RoboDK station: kr30 cnc 071229 table murderer.rdk

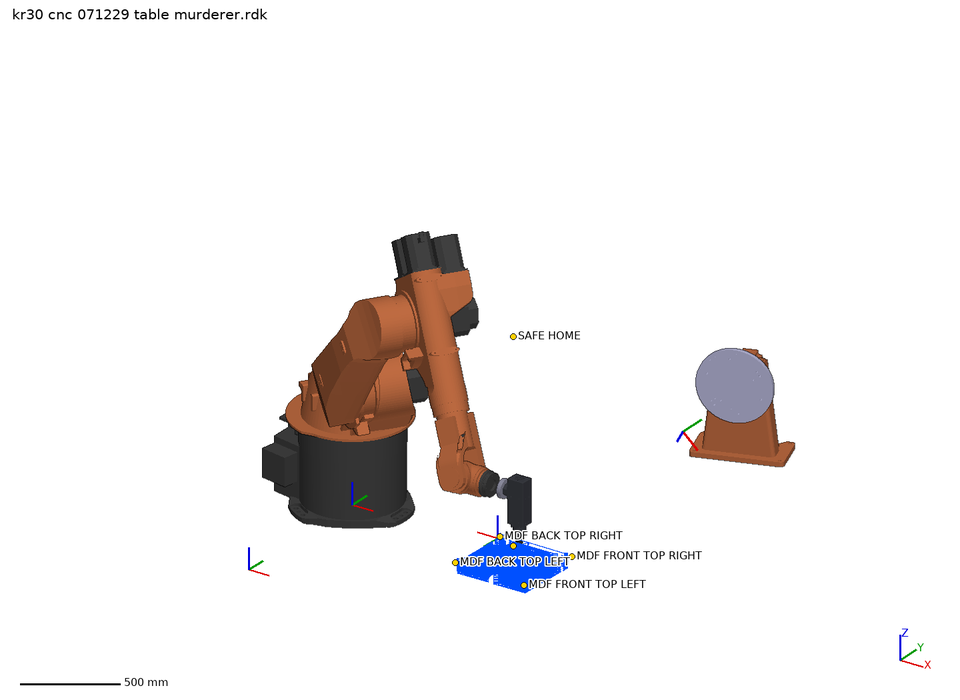
[picture v0: the station drawn from its stored meshes, robots at their saved joint values, targets as dots, program paths as lines]
Station kr30 cnc 071229 table murderer. Poses are relative to the parent item; angles as X-Y-Z fixed-axis rotations.
  - frame GIGASHEEN 7th Axis Base at (0, 1100, 0) mm
    - robot KUKA KP1 MD250: 1 axes, payload 250 kg
        modified DH rows (alpha deg, a mm, theta deg, d mm): 0, 0, 0, 0
        base shift (1750, 1710, 820) mm, rotated rx 0 ry 90 rz -70 deg
        joint limits [-3600] to [3600]; home [0]; saved at [-681.46]
      - frame Reference Rhino at (0, -250, 250) mm
        - object RhinoPart at (0, 0, 0) mm
  - frame GIGASHEEN Base at (0, 2000, 0) mm
    - robot GIGASHEEN (model KUKA KR 30 HA): 6 axes, payload 30 kg, reach 2033 mm, repeatability 0.05 mm, weight 665 kg
        modified DH rows (alpha deg, a mm, theta deg, d mm): 0, 0, 0, 815; -90, 350, 0, 0; 0, 850, -90, 0; -90, 145, 0, 820; 90, 0, 0, 0; -90, 0, 180, 170
        joint limits [-185, -135, -120, -350, -119, -350] to [185, 35, 158, 350, 119, 350]; home [0, -90, 90, 0, 0, 0]; saved at [33.038, -47.483, 104.992, -142.577, 63.826, 162.326]
      - tool 1/2" End Mill TCP, TCP at (337.71, -2.2, 160.57) mm, rotated rx 0 ry 90 rz 0 deg, size 415.8 x 102 x 153.6 mm
    - target MDF BACK TOP LEFT (joint target) at (1355.3, -1043.68, 475.29) mm, rotated rx 179.37 ry 1.37 rz 91.89 deg; joints [27.716, -45.008, 102.25, 116.233, 75.695, -151.59, -681.46] of GIGASHEEN
    - target MDF FRONT TOP LEFT (joint target) at (1780.2, -1054.61, 474.32) mm, rotated rx 179.37 ry 1.37 rz 91.89 deg; joints [22.06, -21.631, 54.581, 104.768, 70.881, -126.376, -681.46] of GIGASHEEN
    - target MDF FRONT TOP RIGHT (joint target) at (1790.65, -653.53, 473.79) mm, rotated rx 179.37 ry 1.37 rz 91.89 deg; joints [10.053, -29.315, 70.245, 98.928, 81.917, -132.341, -681.46] of GIGASHEEN
    - target MDF BACK TOP RIGHT (joint target) at (1365.17, -670.22, 473.91) mm, rotated rx 179.37 ry 1.37 rz 91.89 deg; joints [13.787, -50.344, 113.459, 104.66, 84.215, -154.683, -681.46] of GIGASHEEN
    - target MDF STOCK DEPTH (only use z axis value) (joint target) at (1411.38, -622.96, 416.46) mm, rotated rx 179.37 ry 1.37 rz 91.89 deg; joints [11.502, -45.737, 110.222, 102.707, 85.519, -155.78, -681.46] of GIGASHEEN
    - target SAFE HOME (joint target) at (1411.38, -622.96, 1575.57) mm, rotated rx 179.37 ry 1.37 rz 91.89 deg; joints [11.502, -69.45, 58.776, 88.861, 76.585, -79.989, -681.46] of GIGASHEEN
  - frame Frame 4 at (1373.15, 1298.42, 478.65) mm, rotated rx 1.38 ry 0.62 rz -180 deg
  - machining project Machining Settings: C:/Users/liqui/OneDrive/Documents/GitHub/kuka-fdm/chuck base linearized.apt | rotZ(0) | rotX(0)*rotY(0) | rotz(0)
  - program Machining (9569 instructions, listed below)
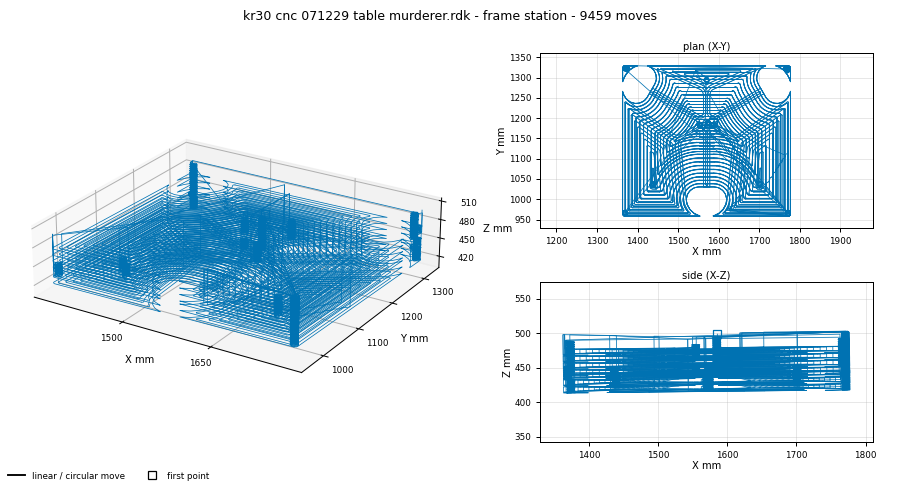
[picture p0: tool path of kr30 cnc 071229 table murderer.rdk in frame station, 9459 of 9459 moves have a stored position in this frame; points joined in program order, loops and branches not executed]

--- program Machining (robot GIGASHEEN) ---
  Accurate (rounding -1 mm)
  Set Ref.: Frame 4
  Set Tool: 1/2" End Mill TCP
  Show 1/2" End Mill TCP
  Print: /'1001'
  Print: /''
  Print: /'Pocket2'
  Set speed (500.0 mm/s)
  Set speed (500.0 mm/s)
  MoveJ 1 to (-212.83, 109.37, 15) mm, rotated rx 180 ry 0 rz 0.01 deg; joints [32.596, -47.797, 105.138, -142.993, 63.549, 162.425]
  MoveL 2 to (-212.83, 109.37, 15) mm, rotated rx 180 ry 0 rz 0.01 deg; joints [32.596, -47.797, 105.138, -142.993, 63.549, 162.425]
  MoveL 3 to (-212.83, 109.37, 15) mm, rotated rx 180 ry 0 rz 0.01 deg; joints [32.596, -47.797, 105.138, -142.993, 63.549, 162.425]
  Set speed (500.0 mm/s)
  MoveL 4 to (-212.83, 109.37, 11.77) mm, rotated rx 180 ry 0 rz 0.01 deg; joints [32.598, -47.633, 105.136, -143.039, 63.679, 162.532]
  Set speed (100.0 mm/s)
  MoveL 5 to (-212.67, 109.35, 11.15) mm, rotated rx -180 ry 0 rz 0.01 deg; joints [32.601, -47.608, 105.149, -143.047, 63.71, 162.556]
  MoveL 6 to (-212.22, 109.32, 10.68) mm, rotated rx -180 ry 0 rz 0.01 deg; joints [32.61, -47.602, 105.184, -143.05, 63.746, 162.58]
  MoveL 7 to (-211.61, 109.34, 10.5) mm, rotated rx 180 ry 0 rz 0.01 deg; joints [32.623, -47.616, 105.231, -143.046, 63.777, 162.596]
  MoveL 8 to (-206.37, 113.36, 10.26) mm, rotated rx -180 ry 0 rz 0.01 deg; joints [32.864, -47.707, 105.436, -142.826, 63.946, 162.558]
  MoveL 9 to (-207.96, 119.77, 10.01) mm, rotated rx -180 ry 0 rz 0.01 deg; joints [33.038, -47.483, 104.992, -142.577, 63.826, 162.326]
  MoveL 10 to (-214.47, 120.88, 9.77) mm, rotated rx -180 ry 0 rz 0.01 deg; joints [32.938, -47.198, 104.43, -142.6, 63.574, 162.187]
  MoveL 11 to (-218.1, 115.37, 9.52) mm, rotated rx -180 ry 0 rz 0.01 deg; joints [32.685, -47.178, 104.424, -142.871, 63.502, 162.318]
  MoveL 12 to (-214.5, 109.83, 9.28) mm, rotated rx 180 ry 0 rz 0.01 deg; joints [32.58, -47.432, 104.981, -143.072, 63.71, 162.572]
  MoveL 13 to (-207.98, 110.91, 9.04) mm, rotated rx 180 ry 0 rz 0.01 deg; joints [32.751, -47.641, 105.433, -142.963, 63.959, 162.653]
  MoveL 14 to (-206.36, 117.31, 8.79) mm, rotated rx 180 ry 0 rz 0.01 deg; joints [32.993, -47.539, 105.238, -142.681, 63.962, 162.476]
  MoveL 15 to (-211.58, 121.36, 8.55) mm, rotated rx 180 ry 0 rz 0.01 deg; joints [33.014, -47.234, 104.629, -142.568, 63.728, 162.261]
  MoveL 16 to (-217.38, 118.21, 8.3) mm, rotated rx -180 ry 0 rz 0.01 deg; joints [32.792, -47.076, 104.336, -142.762, 63.548, 162.276]
  MoveL 17 to (-216.81, 111.63, 8.06) mm, rotated rx 180 ry 0 rz 0.01 deg; joints [32.591, -47.24, 104.709, -143.037, 63.65, 162.513]
  MoveL 18 to (-210.56, 109.51, 7.82) mm, rotated rx 180 ry 0 rz 0.01 deg; joints [32.652, -47.514, 105.301, -143.066, 63.924, 162.697]
  MoveL 19 to (-206.11, 114.39, 7.57) mm, rotated rx -180 ry 0 rz 0.01 deg; joints [32.904, -47.555, 105.402, -142.818, 64.052, 162.618]
  MoveL 20 to (-208.8, 120.42, 7.33) mm, rotated rx 180 ry 0 rz 0.01 deg; joints [33.043, -47.299, 104.891, -142.597, 63.894, 162.38]
  MoveL 21 to (-215.4, 120.37, 7.08) mm, rotated rx 180 ry 0 rz 0.01 deg; joints [32.903, -47.038, 104.379, -142.669, 63.649, 162.277]
  MoveL 22 to (-218.01, 114.3, 6.84) mm, rotated rx 180 ry 0 rz 0.01 deg; joints [32.654, -47.07, 104.481, -142.953, 63.623, 162.444]
  MoveL 23 to (-213.49, 109.49, 6.6) mm, rotated rx -180 ry 0 rz 0.01 deg; joints [32.591, -47.342, 105.073, -143.114, 63.86, 162.689]
  MoveL 24 to (-207.26, 111.7, 6.35) mm, rotated rx 180 ry 0 rz 0.01 deg; joints [32.793, -47.512, 105.446, -142.961, 64.085, 162.728]
  MoveL 25 to (-206.79, 118.29, 6.11) mm, rotated rx 180 ry 0 rz 0.01 deg; joints [33.017, -47.363, 105.152, -142.683, 64.042, 162.526]
  MoveL 26 to (-212.64, 121.36, 5.86) mm, rotated rx -180 ry 0 rz 0.01 deg; joints [32.993, -47.058, 104.543, -142.617, 63.794, 162.332]
  MoveL 27 to (-217.8, 117.23, 5.62) mm, rotated rx 180 ry 0 rz 0.01 deg; joints [32.753, -46.947, 104.349, -142.846, 63.648, 162.39]
  MoveL 28 to (-216.08, 110.85, 5.37) mm, rotated rx -180 ry 0 rz 0.01 deg; joints [32.582, -47.15, 104.802, -143.1, 63.793, 162.64]
  MoveL 29 to (-209.55, 109.87, 5.13) mm, rotated rx -180 ry 0 rz 0.01 deg; joints [32.686, -47.407, 105.358, -143.078, 64.066, 162.791]
  MoveL 30 to (-206.03, 115.46, 4.89) mm, rotated rx 180 ry 0 rz 0.01 deg; joints [32.942, -47.396, 105.351, -142.811, 64.151, 162.673]
  MoveL 31 to (-209.74, 120.92, 4.64) mm, rotated rx 180 ry 0 rz 0.01 deg; joints [33.04, -47.115, 104.789, -142.624, 63.958, 162.437]
  MoveL 32 to (-216.24, 119.71, 4.4) mm, rotated rx -180 ry 0 rz 0.01 deg; joints [32.866, -46.886, 104.344, -142.743, 63.73, 162.374]
  MoveL 33 to (-217.73, 113.27, 4.15) mm, rotated rx -180 ry 0 rz 0.01 deg; joints [32.628, -46.968, 104.55, -143.032, 63.752, 162.571]
  MoveL 34 to (-212.43, 109.33, 3.91) mm, rotated rx 180 ry 0 rz 0.01 deg; joints [32.61, -47.248, 105.159, -143.147, 64.009, 162.8]
  MoveL 35 to (-206.69, 112.6, 3.67) mm, rotated rx 180 ry 0 rz 0.01 deg; joints [32.836, -47.375, 105.441, -142.954, 64.205, 162.797]
  MoveL 36 to (-207.39, 119.17, 3.42) mm, rotated rx 180 ry 0 rz 0.01 deg; joints [33.034, -47.182, 105.057, -142.69, 64.116, 162.576]
  MoveL 37 to (-213.69, 121.16, 3.18) mm, rotated rx 180 ry 0 rz 0.01 deg; joints [32.966, -46.886, 104.468, -142.674, 63.861, 162.41]
  MoveL 38 to (-218.04, 116.19, 2.93) mm, rotated rx 180 ry 0 rz 0.01 deg; joints [32.716, -46.826, 104.378, -142.93, 63.756, 162.509]
  MoveL 39 to (-215.23, 110.21, 2.69) mm, rotated rx -180 ry 0 rz 0.01 deg; joints [32.581, -47.06, 104.896, -143.156, 63.94, 162.764]
  MoveL 40 to (-208.62, 110.4, 2.45) mm, rotated rx -180 ry 0 rz 0.01 deg; joints [32.724, -47.291, 105.399, -143.084, 64.203, 162.877]
  MoveL 41 to (-206.15, 116.52, 2.2) mm, rotated rx -180 ry 0 rz 0.01 deg; joints [32.975, -47.229, 105.285, -142.805, 64.242, 162.725]
  MoveL 42 to (-210.76, 121.24, 1.96) mm, rotated rx -180 ry 0 rz 0.01 deg; joints [33.031, -46.932, 104.689, -142.658, 64.021, 162.498]
  MoveL 43 to (-216.94, 118.9, 1.71) mm, rotated rx -180 ry 0 rz 0.01 deg; joints [32.827, -46.742, 104.326, -142.822, 63.817, 162.477]
  MoveL 44 to (-217.27, 112.31, 1.47) mm, rotated rx 180 ry 0 rz 0.01 deg; joints [32.607, -46.871, 104.63, -143.105, 63.886, 162.699]
  MoveL 45 to (-211.36, 109.36, 1.23) mm, rotated rx -180 ry 0 rz 0.01 deg; joints [32.634, -47.15, 105.236, -143.173, 64.157, 162.905]
  MoveL 46 to (-206.29, 113.59, 0.98) mm, rotated rx 180 ry 0 rz 0.01 deg; joints [32.878, -47.229, 105.418, -142.946, 64.316, 162.86]
  MoveL 47 to (-208.14, 119.93, 0.74) mm, rotated rx 180 ry 0 rz 0.01 deg; joints [33.044, -46.999, 104.957, -142.703, 64.185, 162.626]
  MoveL 48 to (-214.69, 120.78, 0.49) mm, rotated rx -180 ry 0 rz 0.01 deg; joints [32.935, -46.721, 104.404, -142.738, 63.932, 162.494]
  MoveL 49 to (-218.09, 115.12, 0.25) mm, rotated rx -180 ry 0 rz 0.01 deg; joints [32.682, -46.713, 104.423, -143.012, 63.872, 162.632]
  MoveL 50 to (-214.27, 109.74, 0.01) mm, rotated rx 180 ry 0 rz 0.01 deg; joints [32.587, -46.969, 104.989, -143.203, 64.089, 162.883]
  MoveL 51 to (-207.8, 111.08, -0.24) mm, rotated rx 180 ry 0 rz 0.01 deg; joints [32.765, -47.168, 105.424, -143.084, 64.334, 162.957]
  MoveL 52 to (-206.44, 117.54, -0.48) mm, rotated rx 180 ry 0 rz 0.01 deg; joints [33.003, -47.056, 105.206, -142.802, 64.325, 162.775]
  MoveL 53 to (-211.82, 121.38, -0.73) mm, rotated rx 180 ry 0 rz 0.01 deg; joints [33.015, -46.752, 104.595, -142.701, 64.085, 162.563]
  MoveL 54 to (-217.49, 117.99, -0.97) mm, rotated rx -180 ry 0 rz 0.01 deg; joints [32.788, -46.606, 104.324, -142.903, 63.912, 162.586]
  MoveL 55 to (-216.66, 111.44, -1.21) mm, rotated rx -180 ry 0 rz 0.01 deg; joints [32.593, -46.778, 104.716, -143.173, 64.026, 162.826]
  MoveL 56 to (-210.32, 109.58, -1.46) mm, rotated rx -180 ry 0 rz 0.01 deg; joints [32.665, -47.046, 105.302, -143.19, 64.302, 163.004]
  MoveL 57 to (-206.07, 114.63, -1.7) mm, rotated rx 180 ry 0 rz 0.01 deg; joints [32.918, -47.075, 105.378, -142.937, 64.42, 162.917]
  MoveL 58 to (-209.01, 120.55, -1.95) mm, rotated rx 180 ry 0 rz 0.01 deg; joints [33.048, -46.815, 104.853, -142.723, 64.251, 162.679]
  MoveL 59 to (-215.6, 120.23, -2.19) mm, rotated rx -180 ry 0 rz 0.01 deg; joints [32.9, -46.562, 104.356, -142.807, 64.008, 162.584]
  MoveL 60 to (-217.96, 114.06, -2.43) mm, rotated rx 180 ry 0 rz 0.01 deg; joints [32.652, -46.605, 104.481, -143.093, 63.995, 162.757]
  MoveL 61 to (-213.25, 109.44, -2.68) mm, rotated rx -180 ry 0 rz 0.01 deg; joints [32.6, -46.877, 105.079, -143.242, 64.239, 162.998]
  MoveL 62 to (-207.12, 111.9, -2.92) mm, rotated rx -180 ry 0 rz 0.01 deg; joints [32.808, -47.036, 105.431, -143.079, 64.459, 163.03]
  MoveL 63 to (-206.92, 118.5, -3.17) mm, rotated rx -180 ry 0 rz 0.01 deg; joints [33.026, -46.878, 105.116, -142.804, 64.403, 162.823]
  MoveL 64 to (-212.89, 121.33, -3.41) mm, rotated rx 180 ry 0 rz 0.01 deg; joints [32.992, -46.576, 104.51, -142.751, 64.149, 162.635]
  MoveL 65 to (-217.87, 116.99, -3.65) mm, rotated rx -180 ry 0 rz 0.01 deg; joints [32.749, -46.478, 104.339, -142.986, 64.013, 162.701]
  MoveL 66 to (-215.9, 110.69, -3.9) mm, rotated rx -180 ry 0 rz 0.01 deg; joints [32.586, -46.686, 104.808, -143.233, 64.17, 162.951]
  MoveL 67 to (-209.33, 109.97, -4.14) mm, rotated rx -180 ry 0 rz 0.01 deg; joints [32.7, -46.935, 105.353, -143.199, 64.443, 163.095]
  MoveL 68 to (-206.04, 115.7, -4.39) mm, rotated rx -180 ry 0 rz 0.01 deg; joints [32.954, -46.913, 105.321, -142.929, 64.516, 162.971]
  MoveL 69 to (-209.97, 121.01, -4.63) mm, rotated rx 180 ry 0 rz 0.01 deg; joints [33.044, -46.63, 104.75, -142.751, 64.314, 162.736]
  MoveL 70 to (-216.41, 119.53, -4.87) mm, rotated rx -180 ry 0 rz 0.01 deg; joints [32.862, -46.411, 104.322, -142.882, 64.09, 162.681]
  MoveL 71 to (-217.64, 113.05, -5.12) mm, rotated rx -180 ry 0 rz 0.01 deg; joints [32.627, -46.503, 104.551, -143.169, 64.124, 162.883]
  MoveL 72 to (-212.19, 109.32, -5.36) mm, rotated rx -180 ry 0 rz 0.01 deg; joints [32.62, -46.781, 105.161, -143.273, 64.388, 163.107]
  MoveL 73 to (-206.59, 112.82, -5.61) mm, rotated rx 180 ry 0 rz 0.01 deg; joints [32.85, -46.896, 105.42, -143.071, 64.576, 163.096]
  MoveL 74 to (-207.55, 119.35, -5.85) mm, rotated rx -180 ry 0 rz 0.01 deg; joints [33.042, -46.696, 105.018, -142.812, 64.474, 162.872]
  MoveL 75 to (-213.92, 121.09, -6.1) mm, rotated rx -180 ry 0 rz 0.01 deg; joints [32.964, -46.405, 104.435, -142.808, 64.217, 162.712]
  MoveL 76 to (-218.07, 115.95, -6.34) mm, rotated rx -180 ry 0 rz 0.01 deg; joints [32.713, -46.358, 104.37, -143.068, 64.123, 162.819]
  MoveL 77 to (-215.02, 110.09, -6.58) mm, rotated rx 180 ry 0 rz 0.01 deg; joints [32.587, -46.595, 104.9, -143.286, 64.317, 163.073]
  MoveL 78 to (-208.43, 110.54, -6.83) mm, rotated rx -180 ry 0 rz 0.01 deg; joints [32.738, -46.817, 105.389, -143.202, 64.578, 163.179]
  MoveL 79 to (-206.2, 116.76, -7.07) mm, rotated rx 180 ry 0 rz 0.01 deg; joints [32.987, -46.744, 105.25, -142.923, 64.604, 163.021]
  MoveL 80 to (-211, 121.29, -7.32) mm, rotated rx 180 ry 0 rz 0.01 deg; joints [33.033, -46.447, 104.649, -142.787, 64.376, 162.796]
  MoveL 81 to (-217.08, 118.7, -7.56) mm, rotated rx -180 ry 0 rz 0.01 deg; joints [32.823, -46.268, 104.306, -142.96, 64.178, 162.784]
  MoveL 82 to (-217.15, 112.1, -7.8) mm, rotated rx -180 ry 0 rz 0.01 deg; joints [32.608, -46.406, 104.631, -143.24, 64.26, 163.009]
  MoveL 83 to (-211.12, 109.39, -8.05) mm, rotated rx -180 ry 0 rz 0.01 deg; joints [32.646, -46.68, 105.234, -143.295, 64.535, 163.21]
  MoveL 84 to (-206.23, 113.83, -8.29) mm, rotated rx -180 ry 0 rz 0.01 deg; joints [32.892, -46.748, 105.392, -143.062, 64.684, 163.157]
  MoveL 85 to (-208.33, 120.09, -8.54) mm, rotated rx -180 ry 0 rz 0.01 deg; joints [33.051, -46.512, 104.914, -142.826, 64.541, 162.922]
  MoveL 86 to (-214.91, 120.67, -8.78) mm, rotated rx -180 ry 0 rz 0.01 deg; joints [32.932, -46.241, 104.373, -142.872, 64.288, 162.796]
  MoveL 87 to (-218.08, 114.88, -9.02) mm, rotated rx -180 ry 0 rz 0.01 deg; joints [32.679, -46.244, 104.416, -143.15, 64.24, 162.941]
  MoveL 88 to (-214.04, 109.65, -9.27) mm, rotated rx 180 ry 0 rz 0.01 deg; joints [32.594, -46.503, 104.991, -143.331, 64.466, 163.191]
  MoveL 89 to (-207.64, 111.25, -9.51) mm, rotated rx 180 ry 0 rz 0.01 deg; joints [32.78, -46.691, 105.408, -143.2, 64.707, 163.256]
  MoveL 90 to (-206.54, 117.77, -9.76) mm, rotated rx -180 ry 0 rz 0.01 deg; joints [33.014, -46.569, 105.167, -142.92, 64.685, 163.069]
  MoveL 91 to (-212.06, 121.38, -10) mm, rotated rx -180 ry 0 rz 0.01 deg; joints [33.015, -46.268, 104.555, -142.83, 64.439, 162.862]
  MoveL 92 to (-213.99, 121.38, -10) mm, rotated rx -180 ry 0 rz 0.01 deg; joints [32.975, -46.196, 104.405, -142.85, 64.364, 162.828]
  MoveC 93 to (-215.91, 120.27, -10) mm, rotated rx 180 ry 0 rz 0.01 deg; joints [32.899, -46.15, 104.311, -142.916, 64.301, 162.831] to (-215.92, 118.06, -10) mm, rotated rx -180 ry 0 rz 0.01 deg; joints [32.827, -46.201, 104.423, -143.008, 64.326, 162.905]
  MoveL 94 to (-214.81, 116.14, -10) mm, rotated rx -180 ry 0 rz 0.01 deg; joints [32.788, -46.287, 104.605, -143.077, 64.391, 162.988]
  MoveC 95 to (-213.77, 115.1, -10) mm, rotated rx 180 ry 0 rz 0.01 deg; joints [32.776, -46.35, 104.738, -143.11, 64.444, 163.04] to (-212.35, 114.72, -10) mm, rotated rx 180 ry 0 rz 0.01 deg; joints [32.794, -46.412, 104.868, -143.111, 64.504, 163.077]
  MoveL 96 to (-181.15, 114.72, -10) mm, rotated rx 180 ry 0 rz 0.01 deg; joints [33.456, -47.555, 107.262, -142.767, 65.707, 163.609]
  MoveC 97 to (-179.73, 115.1, -10) mm, rotated rx 180 ry 0 rz 0.01 deg; joints [33.499, -47.597, 107.35, -142.735, 65.756, 163.62] to (-178.69, 116.13, -10) mm, rotated rx -180 ry 0 rz 0.01 deg; joints [33.555, -47.611, 107.377, -142.679, 65.784, 163.604]
  MoveL 98 to (-177.58, 118.05, -10) mm, rotated rx 180 ry 0 rz 0.01 deg; joints [33.642, -47.607, 107.365, -142.587, 65.804, 163.561]
  MoveC 99 to (-177.58, 120.27, -10) mm, rotated rx -180 ry 0 rz 0.01 deg; joints [33.714, -47.556, 107.253, -142.495, 65.778, 163.489] to (-179.5, 121.38, -10) mm, rotated rx -180 ry 0 rz 0.01 deg; joints [33.709, -47.461, 107.052, -142.471, 65.692, 163.42]
  MoveL 100 to (-212.06, 121.38, -10) mm, rotated rx -180 ry 0 rz 0.01 deg; joints [33.015, -46.268, 104.555, -142.83, 64.439, 162.862]
  MoveC 101 to (-215.55, 122.47, -10) mm, rotated rx 180 ry 0 rz 0.01 deg; joints [32.977, -46.112, 104.229, -142.82, 64.29, 162.765] to (-217.79, 125.34, -10) mm, rotated rx -180 ry 0 rz 0.01 deg; joints [33.023, -45.961, 103.908, -142.723, 64.17, 162.63]
  MoveC 102 to (-219.97, 128.24, -10) mm, rotated rx 180 ry 0 rz 0.01 deg; joints [33.07, -45.812, 103.59, -142.624, 64.051, 162.494] to (-223.36, 129.52, -10) mm, rotated rx 180 ry 0 rz 0.01 deg; joints [33.04, -45.654, 103.259, -142.603, 63.904, 162.391]
  MoveC 103 to (-226.44, 129.78, -10) mm, rotated rx -180 ry 0 rz 0.01 deg; joints [32.985, -45.532, 103.004, -142.622, 63.78, 162.327] to (-229.51, 130.08, -10) mm, rotated rx -180 ry 0 rz 0.01 deg; joints [32.931, -45.409, 102.747, -142.639, 63.656, 162.262]
  MoveC 104 to (-231.31, 129.16, -10) mm, rotated rx -180 ry 0 rz 0.01 deg; joints [32.865, -45.362, 102.651, -142.694, 63.595, 162.26] to (-231.22, 127.14, -10) mm, rotated rx 180 ry 0 rz 0.01 deg; joints [32.802, -45.413, 102.762, -142.778, 63.622, 162.331]
  MoveC 105 to (-228.51, 123.21, -10) mm, rotated rx 180 ry 0 rz 0.01 deg; joints [32.733, -45.608, 103.175, -142.916, 63.773, 162.511] to (-225.92, 119.21, -10) mm, rotated rx 180 ry 0 rz 0.01 deg; joints [32.657, -45.799, 103.581, -143.059, 63.921, 162.691]
  MoveC 106 to (-223.44, 115.14, -10) mm, rotated rx 180 ry 0 rz 0.01 deg; joints [32.578, -45.987, 103.981, -143.205, 64.065, 162.87] to (-221.02, 111.03, -10) mm, rotated rx -180 ry 0 rz 0.01 deg; joints [32.495, -46.173, 104.375, -143.353, 64.206, 163.048]
  MoveC 107 to (-217.92, 107.92, -10) mm, rotated rx 180 ry 0 rz 0.01 deg; joints [32.458, -46.36, 104.773, -143.452, 64.363, 163.204] to (-213.68, 106.78, -10) mm, rotated rx 180 ry 0 rz 0.01 deg; joints [32.509, -46.544, 105.16, -143.457, 64.542, 163.315]
  MoveL 108 to (-179.84, 106.78, -10) mm, rotated rx 180 ry 0 rz 0.01 deg; joints [33.224, -47.784, 107.756, -143.082, 65.848, 163.886]
  MoveC 109 to (-175.59, 107.92, -10) mm, rotated rx 180 ry 0 rz 0.01 deg; joints [33.353, -47.911, 108.021, -142.983, 65.997, 163.92] to (-172.48, 111.03, -10) mm, rotated rx -180 ry 0 rz 0.01 deg; joints [33.523, -47.951, 108.1, -142.817, 66.079, 163.872]
  MoveC 110 to (-170.06, 115.13, -10) mm, rotated rx 180 ry 0 rz 0.01 deg; joints [33.71, -47.944, 108.076, -142.617, 66.123, 163.78] to (-167.6, 119.21, -10) mm, rotated rx 180 ry 0 rz 0.01 deg; joints [33.898, -47.938, 108.057, -142.418, 66.168, 163.69]
  MoveC 111 to (-165.03, 123.22, -10) mm, rotated rx 180 ry 0 rz 0.01 deg; joints [34.086, -47.937, 108.047, -142.22, 66.219, 163.603] to (-162.31, 127.14, -10) mm, rotated rx 180 ry 0 rz 0.01 deg; joints [34.273, -47.942, 108.051, -142.024, 66.275, 163.522]
  MoveC 112 to (-162.21, 129.16, -10) mm, rotated rx 180 ry 0 rz 0.01 deg; joints [34.342, -47.899, 107.956, -141.94, 66.256, 163.458] to (-164.01, 130.09, -10) mm, rotated rx -180 ry 0 rz 0.01 deg; joints [34.332, -47.813, 107.775, -141.924, 66.177, 163.398]
  MoveC 113 to (-167.84, 129.69, -10) mm, rotated rx -180 ry 0 rz 0.01 deg; joints [34.234, -47.685, 107.508, -141.987, 66.038, 163.346] to (-171.67, 129.27, -10) mm, rotated rx 180 ry 0 rz 0.01 deg; joints [34.136, -47.558, 107.243, -142.051, 65.898, 163.295]
  MoveC 114 to (-175.51, 128.94, -10) mm, rotated rx -180 ry 0 rz 0.01 deg; joints [34.041, -47.428, 106.97, -142.111, 65.756, 163.241] to (-179.36, 128.83, -10) mm, rotated rx 180 ry 0 rz 0.01 deg; joints [33.954, -47.292, 106.685, -142.161, 65.611, 163.179]
  MoveL 115 to (-205.63, 128.84, -10) mm, rotated rx -180 ry 0 rz 0.01 deg; joints [33.39, -46.332, 104.676, -142.453, 64.603, 162.727]
  MoveC 116 to (-214.5, 129.01, -10) mm, rotated rx -180 ry 0 rz 0.01 deg; joints [33.209, -45.998, 103.978, -142.537, 64.256, 162.565] to (-223.36, 129.52, -10) mm, rotated rx -180 ry 0 rz 0.01 deg; joints [33.04, -45.654, 103.259, -142.603, 63.904, 162.391]
  MoveC 117 to (-226.59, 130.78, -10) mm, rotated rx 180 ry 0 rz 0.01 deg; joints [33.014, -45.502, 102.941, -142.582, 63.763, 162.29] to (-228.56, 133.63, -10) mm, rotated rx -180 ry 0 rz 0.01 deg; joints [33.063, -45.36, 102.639, -142.482, 63.652, 162.159]
  MoveC 118 to (-230.49, 136.49, -10) mm, rotated rx -180 ry 0 rz 0.01 deg; joints [33.114, -45.219, 102.34, -142.38, 63.544, 162.026] to (-233.65, 137.88, -10) mm, rotated rx -180 ry 0 rz 0.01 deg; joints [33.093, -45.066, 102.018, -142.351, 63.403, 161.922]
  MoveC 119 to (-239.01, 138.68, -10) mm, rotated rx -180 ry 0 rz 0.01 deg; joints [33.008, -44.842, 101.55, -142.365, 63.182, 161.796] to (-244.35, 139.65, -10) mm, rotated rx 180 ry 0 rz 0.01 deg; joints [32.93, -44.614, 101.074, -142.371, 62.958, 161.664]
  MoveC 120 to (-245.19, 139.83, -10) mm, rotated rx 180 ry 0 rz 0.01 deg; joints [32.918, -44.577, 100.997, -142.371, 62.923, 161.642] to (-246.02, 140.03, -10) mm, rotated rx 180 ry 0 rz 0.01 deg; joints [32.908, -44.54, 100.92, -142.37, 62.888, 161.62]
  MoveC 121 to (-246.85, 140.23, -10) mm, rotated rx -180 ry 0 rz 0.01 deg; joints [32.897, -44.504, 100.843, -142.368, 62.852, 161.597] to (-247.69, 140.41, -10) mm, rotated rx 180 ry 0 rz 0.01 deg; joints [32.886, -44.467, 100.766, -142.368, 62.817, 161.576]
  MoveC 122 to (-249.42, 139.63, -10) mm, rotated rx -180 ry 0 rz 0.01 deg; joints [32.826, -44.419, 100.667, -142.415, 62.756, 161.57] to (-249.25, 137.73, -10) mm, rotated rx -180 ry 0 rz 0.01 deg; joints [32.77, -44.471, 100.779, -142.493, 62.784, 161.639]
  MoveC 123 to (-245.42, 133.29, -10) mm, rotated rx 180 ry 0 rz 0.01 deg; joints [32.708, -44.725, 101.316, -142.647, 62.988, 161.863] to (-241.53, 128.89, -10) mm, rotated rx 180 ry 0 rz 0.01 deg; joints [32.647, -44.979, 101.852, -142.798, 63.193, 162.084]
  MoveC 124 to (-237.77, 124.39, -10) mm, rotated rx -180 ry 0 rz 0.01 deg; joints [32.58, -45.229, 102.382, -142.953, 63.394, 162.306] to (-234.3, 119.65, -10) mm, rotated rx 180 ry 0 rz 0.01 deg; joints [32.5, -45.472, 102.897, -143.12, 63.585, 162.527]
  MoveC 125 to (-231.84, 115.78, -10) mm, rotated rx -180 ry 0 rz 0.01 deg; joints [32.426, -45.656, 103.287, -143.259, 63.726, 162.701] to (-229.63, 111.75, -10) mm, rotated rx 180 ry 0 rz 0.01 deg; joints [32.341, -45.832, 103.663, -143.407, 63.859, 162.874]
  MoveC 126 to (-227.51, 107.68, -10) mm, rotated rx -180 ry 0 rz 0.01 deg; joints [32.254, -46.006, 104.033, -143.557, 63.989, 163.046] to (-225.27, 103.68, -10) mm, rotated rx 180 ry 0 rz 0.01 deg; joints [32.169, -46.181, 104.407, -143.703, 64.123, 163.216]
  MoveC 127 to (-222.17, 100.57, -10) mm, rotated rx 180 ry 0 rz 0.01 deg; joints [32.132, -46.369, 104.804, -143.803, 64.28, 163.372] to (-217.92, 99.43, -10) mm, rotated rx 180 ry 0 rz 0.01 deg; joints [32.182, -46.553, 105.192, -143.808, 64.46, 163.482]
  MoveL 128 to (-175.6, 99.43, -10) mm, rotated rx -180 ry 0 rz 0.01 deg; joints [33.073, -48.102, 108.438, -143.337, 66.094, 164.191]
  MoveC 129 to (-171.35, 100.57, -10) mm, rotated rx 180 ry 0 rz 0.01 deg; joints [33.202, -48.229, 108.702, -143.237, 66.243, 164.224] to (-168.24, 103.68, -10) mm, rotated rx -180 ry 0 rz 0.01 deg; joints [33.373, -48.27, 108.783, -143.07, 66.324, 164.176]
  MoveC 130 to (-164.24, 110.52, -10) mm, rotated rx -180 ry 0 rz 0.01 deg; joints [33.687, -48.257, 108.743, -142.736, 66.396, 164.024] to (-160.18, 117.33, -10) mm, rotated rx 180 ry 0 rz 0.01 deg; joints [34, -48.245, 108.705, -142.403, 66.47, 163.873]
  MoveC 131 to (-155.83, 123.97, -10) mm, rotated rx 180 ry 0 rz 0.01 deg; joints [34.314, -48.245, 108.694, -142.073, 66.555, 163.732] to (-150.99, 130.25, -10) mm, rotated rx -180 ry 0 rz 0.01 deg; joints [34.628, -48.269, 108.733, -141.751, 66.662, 163.609]
  MoveC 132 to (-149.35, 132.16, -10) mm, rotated rx 180 ry 0 rz 0.01 deg; joints [34.727, -48.282, 108.757, -141.652, 66.701, 163.575] to (-147.65, 134.01, -10) mm, rotated rx -180 ry 0 rz 0.01 deg; joints [34.826, -48.299, 108.787, -141.553, 66.743, 163.543]
  MoveC 133 to (-145.94, 135.85, -10) mm, rotated rx 180 ry 0 rz 0.01 deg; joints [34.924, -48.315, 108.819, -141.455, 66.785, 163.512] to (-144.26, 137.72, -10) mm, rotated rx -180 ry 0 rz 0.01 deg; joints [35.023, -48.33, 108.847, -141.356, 66.825, 163.479]
  MoveC 134 to (-144.06, 139.61, -10) mm, rotated rx 180 ry 0 rz 0.01 deg; joints [35.089, -48.292, 108.764, -141.276, 66.81, 163.421] to (-145.78, 140.42, -10) mm, rotated rx 180 ry 0 rz 0.01 deg; joints [35.076, -48.213, 108.596, -141.266, 66.737, 163.366]
  MoveC 135 to (-154.12, 138.92, -10) mm, rotated rx 180 ry 0 rz 0.01 deg; joints [34.839, -47.955, 108.058, -141.435, 66.444, 163.276] to (-162.48, 137.5, -10) mm, rotated rx -180 ry 0 rz 0.01 deg; joints [34.606, -47.693, 107.51, -141.599, 66.149, 163.181]
  MoveC 136 to (-170.89, 136.46, -10) mm, rotated rx -180 ry 0 rz 0.01 deg; joints [34.386, -47.417, 106.933, -141.745, 65.844, 163.073] to (-179.36, 136.12, -10) mm, rotated rx -180 ry 0 rz 0.01 deg; joints [34.189, -47.12, 106.313, -141.86, 65.527, 162.94]
  MoveL 137 to (-211.94, 136.31, -10) mm, rotated rx -180 ry 0 rz 0.01 deg; joints [33.495, -45.921, 103.804, -142.207, 64.272, 162.365]
  MoveC 138 to (-222.82, 136.77, -10) mm, rotated rx -180 ry 0 rz 0.01 deg; joints [33.282, -45.502, 102.93, -142.296, 63.842, 162.156] to (-233.65, 137.88, -10) mm, rotated rx -180 ry 0 rz 0.01 deg; joints [33.093, -45.066, 102.018, -142.351, 63.403, 161.922]
  MoveC 139 to (-236.39, 139.14, -10) mm, rotated rx -180 ry 0 rz 0.01 deg; joints [33.076, -44.931, 101.735, -142.323, 63.281, 161.828] to (-237.97, 141.71, -10) mm, rotated rx 180 ry 0 rz 0.01 deg; joints [33.125, -44.809, 101.477, -142.23, 63.189, 161.711]
  MoveC 140 to (-239.5, 144.29, -10) mm, rotated rx -180 ry 0 rz 0.01 deg; joints [33.175, -44.688, 101.22, -142.135, 63.099, 161.594] to (-242.17, 145.66, -10) mm, rotated rx 180 ry 0 rz 0.01 deg; joints [33.163, -44.553, 100.935, -142.101, 62.977, 161.497]
  MoveC 141 to (-243.73, 145.98, -10) mm, rotated rx -180 ry 0 rz 0.01 deg; joints [33.141, -44.485, 100.794, -142.101, 62.911, 161.457] to (-245.29, 146.31, -10) mm, rotated rx 180 ry 0 rz 0.01 deg; joints [33.119, -44.417, 100.651, -142.1, 62.845, 161.416]
  MoveC 142 to (-260.07, 150.25, -10) mm, rotated rx -180 ry 0 rz 0.01 deg; joints [32.943, -43.747, 99.251, -142.054, 62.208, 160.998] to (-274.43, 155.48, -10) mm, rotated rx 180 ry 0 rz 0.01 deg; joints [32.817, -43.05, 97.796, -141.937, 61.566, 160.532]
  MoveC 143 to (-275.99, 154.95, -10) mm, rotated rx 180 ry 0 rz 0.01 deg; joints [32.77, -43.002, 97.695, -141.97, 61.508, 160.521] to (-275.66, 153.34, -10) mm, rotated rx -180 ry 0 rz 0.01 deg; joints [32.727, -43.055, 97.808, -142.036, 61.54, 160.585]
  MoveC 144 to (-256.3, 136, -10) mm, rotated rx -180 ry 0 rz 0.01 deg; joints [32.573, -44.239, 100.3, -142.623, 62.521, 161.567] to (-239.99, 115.76, -10) mm, rotated rx -180 ry 0 rz 0.01 deg; joints [32.26, -45.346, 102.641, -143.335, 63.403, 162.556]
  MoveC 145 to (-237.06, 111.16, -10) mm, rotated rx -180 ry 0 rz 0.01 deg; joints [32.171, -45.564, 103.104, -143.501, 63.572, 162.762] to (-234.44, 106.38, -10) mm, rotated rx -180 ry 0 rz 0.01 deg; joints [32.07, -45.773, 103.55, -143.678, 63.73, 162.967]
  MoveC 146 to (-231.91, 101.55, -10) mm, rotated rx 180 ry 0 rz 0.01 deg; joints [31.965, -45.979, 103.989, -143.857, 63.885, 163.171] to (-229.25, 96.79, -10) mm, rotated rx -180 ry 0 rz 0.01 deg; joints [31.864, -46.188, 104.432, -144.031, 64.044, 163.373]
  MoveC 147 to (-226.15, 93.68, -10) mm, rotated rx -180 ry 0 rz 0.01 deg; joints [31.826, -46.374, 104.829, -144.131, 64.201, 163.528] to (-221.9, 92.54, -10) mm, rotated rx 180 ry 0 rz 0.01 deg; joints [31.875, -46.559, 105.217, -144.137, 64.382, 163.637]
  MoveL 148 to (-171.62, 92.54, -10) mm, rotated rx 180 ry 0 rz 0.01 deg; joints [32.93, -48.399, 109.074, -143.575, 66.325, 164.473]
  MoveC 149 to (-167.37, 93.68, -10) mm, rotated rx 180 ry 0 rz 0.01 deg; joints [33.06, -48.525, 109.337, -143.475, 66.473, 164.506] to (-164.26, 96.79, -10) mm, rotated rx -180 ry 0 rz 0.01 deg; joints [33.231, -48.566, 109.418, -143.306, 66.554, 164.459]
  MoveL 150 to (-155.69, 111.78, -10) mm, rotated rx -180 ry 0 rz 0.01 deg; joints [33.917, -48.531, 109.316, -142.575, 66.703, 164.124]
  MoveC 151 to (-151.1, 119.11, -10) mm, rotated rx 180 ry 0 rz 0.01 deg; joints [34.261, -48.524, 109.289, -142.212, 66.789, 163.966] to (-145.88, 125.99, -10) mm, rotated rx -180 ry 0 rz 0.01 deg; joints [34.604, -48.548, 109.327, -141.86, 66.903, 163.831]
  MoveC 152 to (-139.41, 133.39, -10) mm, rotated rx -180 ry 0 rz 0.01 deg; joints [34.993, -48.601, 109.424, -141.469, 67.055, 163.7] to (-132.6, 140.47, -10) mm, rotated rx -180 ry 0 rz 0.01 deg; joints [35.38, -48.671, 109.557, -141.086, 67.223, 163.583]
  MoveC 153 to (-125.4, 147.16, -10) mm, rotated rx -180 ry 0 rz 0.01 deg; joints [35.764, -48.76, 109.733, -140.712, 67.407, 163.485] to (-117.79, 153.38, -10) mm, rotated rx 180 ry 0 rz 0.01 deg; joints [36.144, -48.872, 109.956, -140.35, 67.611, 163.408]
  MoveC 154 to (-117.47, 154.99, -10) mm, rotated rx -180 ry 0 rz 0.01 deg; joints [36.203, -48.844, 109.894, -140.28, 67.603, 163.361] to (-119.03, 155.51, -10) mm, rotated rx 180 ry 0 rz 0.01 deg; joints [36.183, -48.778, 109.755, -140.281, 67.54, 163.318]
  MoveC 155 to (-144.72, 147.15, -10) mm, rotated rx 180 ry 0 rz 0.01 deg; joints [35.318, -48.09, 108.325, -140.975, 66.697, 163.164] to (-171.45, 143.25, -10) mm, rotated rx -180 ry 0 rz 0.01 deg; joints [34.592, -47.236, 106.542, -141.472, 65.744, 162.839]
  MoveL 156 to (-214.92, 143.01, -10) mm, rotated rx -180 ry 0 rz 0.01 deg; joints [33.646, -45.649, 103.226, -141.959, 64.08, 162.086]
  MoveC 157 to (-228.61, 143.68, -10) mm, rotated rx 180 ry 0 rz 0.01 deg; joints [33.38, -45.118, 102.117, -142.063, 63.536, 161.815] to (-242.17, 145.66, -10) mm, rotated rx 180 ry 0 rz 0.01 deg; joints [33.163, -44.553, 100.935, -142.101, 62.977, 161.497]
  MoveC 158 to (-244.83, 147.08, -10) mm, rotated rx 180 ry 0 rz 0.01 deg; joints [33.153, -44.416, 100.648, -142.064, 62.854, 161.398] to (-246.26, 149.74, -10) mm, rotated rx -180 ry 0 rz 0.01 deg; joints [33.207, -44.296, 100.394, -141.965, 62.767, 161.278]
  MoveC 159 to (-247.64, 152.41, -10) mm, rotated rx 180 ry 0 rz 0.01 deg; joints [33.262, -44.177, 100.142, -141.865, 62.682, 161.159] to (-250.24, 153.93, -10) mm, rotated rx 180 ry 0 rz 0.01 deg; joints [33.256, -44.039, 99.853, -141.822, 62.561, 161.056]
  MoveC 160 to (-267.07, 159.34, -10) mm, rotated rx -180 ry 0 rz 0.01 deg; joints [33.083, -43.247, 98.196, -141.723, 61.821, 160.539] to (-283.1, 166.79, -10) mm, rotated rx 180 ry 0 rz 0.01 deg; joints [32.992, -42.42, 96.47, -141.516, 61.082, 159.95]
  MoveC 161 to (-285.35, 166.74, -10) mm, rotated rx 180 ry 0 rz 0.01 deg; joints [32.946, -42.331, 96.285, -141.532, 60.991, 159.906] to (-286.46, 164.79, -10) mm, rotated rx 180 ry 0 rz 0.01 deg; joints [32.865, -42.336, 96.298, -141.621, 60.967, 159.955]
  MoveL 162 to (-286.46, 156.66, -10) mm, rotated rx 180 ry 0 rz 0.01 deg; joints [32.616, -42.54, 96.735, -141.966, 61.06, 160.251]
  MoveC 163 to (-285.7, 153.53, -10) mm, rotated rx 180 ry 0 rz 0.01 deg; joints [32.535, -42.648, 96.965, -142.094, 61.127, 160.379] to (-283.59, 151.1, -10) mm, rotated rx 180 ry 0 rz 0.01 deg; joints [32.502, -42.793, 97.269, -142.183, 61.241, 160.508]
  MoveC 164 to (-262.73, 133.3, -10) mm, rotated rx 180 ry 0 rz 0.01 deg; joints [32.36, -44.053, 99.917, -142.787, 62.293, 161.54] to (-245.34, 112.1, -10) mm, rotated rx -180 ry 0 rz 0.01 deg; joints [32.035, -45.226, 102.397, -143.536, 63.231, 162.583]
  MoveC 165 to (-241.98, 106.82, -10) mm, rotated rx 180 ry 0 rz 0.01 deg; joints [31.933, -45.476, 102.929, -143.728, 63.425, 162.82] to (-238.96, 101.32, -10) mm, rotated rx -180 ry 0 rz 0.01 deg; joints [31.816, -45.717, 103.441, -143.932, 63.607, 163.055]
  MoveC 166 to (-236.05, 95.78, -10) mm, rotated rx -180 ry 0 rz 0.01 deg; joints [31.694, -45.953, 103.944, -144.138, 63.786, 163.289] to (-233, 90.31, -10) mm, rotated rx 180 ry 0 rz 0.01 deg; joints [31.577, -46.192, 104.453, -144.34, 63.968, 163.52]
  MoveC 167 to (-229.89, 87.2, -10) mm, rotated rx 180 ry 0 rz 0.01 deg; joints [31.538, -46.378, 104.848, -144.44, 64.127, 163.674] to (-225.65, 86.06, -10) mm, rotated rx -180 ry 0 rz 0.01 deg; joints [31.586, -46.563, 105.237, -144.447, 64.307, 163.783]
  MoveL 168 to (-167.88, 86.06, -10) mm, rotated rx -180 ry 0 rz 0.01 deg; joints [32.794, -48.676, 109.668, -143.799, 66.542, 164.737]
  MoveC 169 to (-163.63, 87.2, -10) mm, rotated rx 180 ry 0 rz 0.01 deg; joints [32.924, -48.802, 109.931, -143.698, 66.689, 164.769] to (-160.52, 90.31, -10) mm, rotated rx -180 ry 0 rz 0.01 deg; joints [33.096, -48.843, 110.013, -143.529, 66.771, 164.722]
  MoveC 170 to (-155.91, 98.38, -10) mm, rotated rx -180 ry 0 rz 0.01 deg; joints [33.467, -48.826, 109.962, -143.134, 66.85, 164.544] to (-151.38, 106.49, -10) mm, rotated rx -180 ry 0 rz 0.01 deg; joints [33.838, -48.803, 109.898, -142.738, 66.926, 164.362]
  MoveC 171 to (-146.5, 114.42, -10) mm, rotated rx -180 ry 0 rz 0.01 deg; joints [34.209, -48.794, 109.863, -142.345, 67.015, 164.19] to (-140.9, 121.84, -10) mm, rotated rx -180 ry 0 rz 0.01 deg; joints [34.581, -48.819, 109.902, -141.964, 67.136, 164.046]
  MoveC 172 to (-133.85, 129.86, -10) mm, rotated rx 180 ry 0 rz 0.01 deg; joints [35.005, -48.877, 110.01, -141.538, 67.302, 163.904] to (-126.38, 137.49, -10) mm, rotated rx 180 ry 0 rz 0.01 deg; joints [35.427, -48.956, 110.162, -141.121, 67.486, 163.782]
  MoveC 173 to (-118.43, 144.61, -10) mm, rotated rx -180 ry 0 rz 0.01 deg; joints [35.845, -49.059, 110.367, -140.717, 67.691, 163.682] to (-109.95, 151.1, -10) mm, rotated rx -180 ry 0 rz 0.01 deg; joints [36.256, -49.193, 110.637, -140.329, 67.922, 163.611]
  MoveC 174 to (-107.82, 153.53, -10) mm, rotated rx 180 ry 0 rz 0.01 deg; joints [36.385, -49.207, 110.661, -140.199, 67.969, 163.567] to (-107.06, 156.67, -10) mm, rotated rx -180 ry 0 rz 0.01 deg; joints [36.505, -49.157, 110.551, -140.06, 67.959, 163.478]
  MoveL 175 to (-107.06, 164.75, -10) mm, rotated rx 180 ry 0 rz 0.01 deg; joints [36.765, -48.961, 110.123, -139.733, 67.863, 163.214]
  MoveC 176 to (-108.17, 166.71, -10) mm, rotated rx -180 ry 0 rz 0.01 deg; joints [36.801, -48.875, 109.94, -139.67, 67.8, 163.131] to (-110.41, 166.76, -10) mm, rotated rx -180 ry 0 rz 0.01 deg; joints [36.749, -48.798, 109.777, -139.701, 67.718, 163.092]
  MoveC 177 to (-124.97, 159.99, -10) mm, rotated rx -180 ry 0 rz 0.01 deg; joints [36.188, -48.465, 109.091, -140.183, 67.271, 163.073] to (-140.21, 154.92, -10) mm, rotated rx -180 ry 0 rz 0.01 deg; joints [35.671, -48.06, 108.25, -140.598, 66.773, 162.984]
  MoveC 178 to (-155.9, 151.52, -10) mm, rotated rx 180 ry 0 rz 0.01 deg; joints [35.204, -47.591, 107.272, -140.941, 66.231, 162.831] to (-171.85, 149.72, -10) mm, rotated rx 180 ry 0 rz 0.01 deg; joints [34.79, -47.066, 106.175, -141.21, 65.654, 162.618]
  MoveL 179 to (-214.91, 149.49, -10) mm, rotated rx 180 ry 0 rz 0.01 deg; joints [33.85, -45.493, 102.888, -141.689, 64.005, 161.865]
  MoveC 180 to (-232.71, 150.61, -10) mm, rotated rx -180 ry 0 rz 0.01 deg; joints [33.513, -44.794, 101.429, -141.811, 63.295, 161.501] to (-250.24, 153.93, -10) mm, rotated rx -180 ry 0 rz 0.01 deg; joints [33.256, -44.039, 99.853, -141.822, 62.561, 161.056]
  MoveC 181 to (-253.51, 155.92, -10) mm, rotated rx 180 ry 0 rz 0.01 deg; joints [33.251, -43.863, 99.483, -141.765, 62.407, 160.924] to (-255.11, 159.41, -10) mm, rotated rx -180 ry 0 rz 0.01 deg; joints [33.327, -43.714, 99.168, -141.631, 62.303, 160.77]
  MoveC 182 to (-256.63, 162.91, -10) mm, rotated rx -180 ry 0 rz 0.01 deg; joints [33.404, -43.568, 98.858, -141.496, 62.202, 160.616] to (-259.75, 165.09, -10) mm, rotated rx 180 ry 0 rz 0.01 deg; joints [33.408, -43.391, 98.487, -141.428, 62.051, 160.477]
  MoveC 183 to (-271.74, 169.87, -10) mm, rotated rx -180 ry 0 rz 0.01 deg; joints [33.312, -42.797, 97.246, -141.312, 61.511, 160.067] to (-283.23, 175.76, -10) mm, rotated rx 180 ry 0 rz 0.01 deg; joints [33.262, -42.187, 95.971, -141.137, 60.975, 159.619]
  MoveC 184 to (-285.29, 177.01, -10) mm, rotated rx 180 ry 0 rz 0.01 deg; joints [33.259, -42.072, 95.731, -141.096, 60.876, 159.53] to (-287.27, 178.38, -10) mm, rotated rx 180 ry 0 rz 0.01 deg; joints [33.261, -41.956, 95.489, -141.05, 60.779, 159.438]
  MoveC 185 to (-289.24, 179.77, -10) mm, rotated rx -180 ry 0 rz 0.01 deg; joints [33.264, -41.841, 95.247, -141.002, 60.682, 159.346] to (-291.23, 181.12, -10) mm, rotated rx 180 ry 0 rz 0.01 deg; joints [33.265, -41.725, 95.005, -140.956, 60.584, 159.254]
  MoveC 186 to (-293.4, 181.21, -10) mm, rotated rx -180 ry 0 rz 0.01 deg; joints [33.225, -41.634, 94.816, -140.964, 60.493, 159.205] to (-294.52, 179.35, -10) mm, rotated rx 180 ry 0 rz 0.01 deg; joints [33.147, -41.637, 94.825, -141.049, 60.468, 159.251]
  MoveL 187 to (-294.52, 153.79, -10) mm, rotated rx 180 ry 0 rz 0.01 deg; joints [32.371, -42.285, 96.212, -142.136, 60.76, 160.191]
  MoveC 188 to (-293.42, 149.39, -10) mm, rotated rx 180 ry 0 rz 0.01 deg; joints [32.257, -42.439, 96.538, -142.316, 60.855, 160.373] to (-290.39, 146.01, -10) mm, rotated rx -180 ry 0 rz 0.01 deg; joints [32.212, -42.646, 96.971, -142.442, 61.019, 160.556]
  MoveC 189 to (-279.46, 137.81, -10) mm, rotated rx 180 ry 0 rz 0.01 deg; joints [32.171, -43.284, 98.31, -142.719, 61.561, 161.063] to (-269.38, 128.59, -10) mm, rotated rx -180 ry 0 rz 0.01 deg; joints [32.08, -43.905, 99.616, -143.036, 62.077, 161.578]
  MoveC 190 to (-260.21, 118.47, -10) mm, rotated rx 180 ry 0 rz 0.01 deg; joints [31.942, -44.503, 100.879, -143.393, 62.562, 162.098] to (-252, 107.56, -10) mm, rotated rx 180 ry 0 rz 0.01 deg; joints [31.756, -45.075, 102.09, -143.785, 63.016, 162.616]
  MoveL 191 to (-237.66, 82.25, -10) mm, rotated rx 180 ry 0 rz 0.01 deg; joints [31.22, -46.194, 104.473, -144.723, 63.874, 163.702]
  MoveC 192 to (-234.55, 79.14, -10) mm, rotated rx -180 ry 0 rz 0.01 deg; joints [31.18, -46.38, 104.868, -144.825, 64.032, 163.855] to (-230.31, 78, -10) mm, rotated rx 180 ry 0 rz 0.01 deg; joints [31.227, -46.566, 105.258, -144.832, 64.214, 163.964]
  MoveL 193 to (-163.23, 78, -10) mm, rotated rx 180 ry 0 rz 0.01 deg; joints [32.623, -49.017, 110.403, -144.077, 66.811, 165.061]
  MoveC 194 to (-158.98, 79.14, -10) mm, rotated rx -180 ry 0 rz 0.01 deg; joints [32.754, -49.143, 110.666, -143.975, 66.958, 165.093] to (-155.87, 82.25, -10) mm, rotated rx -180 ry 0 rz 0.01 deg; joints [32.926, -49.185, 110.748, -143.805, 67.039, 165.047]
  MoveL 195 to (-143.61, 103.31, -10) mm, rotated rx 180 ry 0 rz 0.01 deg; joints [33.905, -49.147, 110.628, -142.766, 67.252, 164.588]
  MoveC 196 to (-136.95, 113.52, -10) mm, rotated rx -180 ry 0 rz 0.01 deg; joints [34.395, -49.147, 110.608, -142.253, 67.38, 164.374] to (-129.34, 123.05, -10) mm, rotated rx -180 ry 0 rz 0.01 deg; joints [34.885, -49.191, 110.683, -141.755, 67.548, 164.195]
  MoveC 197 to (-116.98, 135.38, -10) mm, rotated rx -180 ry 0 rz 0.01 deg; joints [35.577, -49.327, 110.948, -141.073, 67.854, 164.003] to (-103.13, 146, -10) mm, rotated rx 180 ry 0 rz 0.01 deg; joints [36.253, -49.546, 111.388, -140.435, 68.228, 163.887]
  MoveC 198 to (-100.09, 149.35, -10) mm, rotated rx 180 ry 0 rz 0.01 deg; joints [36.435, -49.568, 111.429, -140.252, 68.297, 163.828] to (-98.99, 153.74, -10) mm, rotated rx -180 ry 0 rz 0.01 deg; joints [36.604, -49.499, 111.277, -140.058, 68.284, 163.705]
  MoveL 199 to (-99, 179.3, -10) mm, rotated rx 180 ry 0 rz 0.01 deg; joints [37.424, -48.874, 109.915, -139.026, 67.978, 162.868]
  MoveC 200 to (-100.11, 181.18, -10) mm, rotated rx 180 ry 0 rz 0.01 deg; joints [37.457, -48.79, 109.735, -138.967, 67.916, 162.787] to (-102.29, 181.11, -10) mm, rotated rx 180 ry 0 rz 0.01 deg; joints [37.401, -48.718, 109.584, -139.002, 67.839, 162.753]
  MoveL 201 to (-112.71, 174.51, -10) mm, rotated rx -180 ry 0 rz 0.01 deg; joints [36.941, -48.529, 109.199, -139.421, 67.544, 162.798]
  MoveC 202 to (-118.05, 171.44, -10) mm, rotated rx -180 ry 0 rz 0.01 deg; joints [36.716, -48.423, 108.981, -139.622, 67.387, 162.811] to (-123.62, 168.78, -10) mm, rotated rx -180 ry 0 rz 0.01 deg; joints [36.5, -48.297, 108.722, -139.808, 67.217, 162.805]
  MoveC 203 to (-135.37, 164.38, -10) mm, rotated rx -180 ry 0 rz 0.01 deg; joints [36.085, -47.999, 108.104, -140.148, 66.839, 162.753] to (-147.5, 161.16, -10) mm, rotated rx 180 ry 0 rz 0.01 deg; joints [35.703, -47.654, 107.386, -140.439, 66.43, 162.654]
  MoveC 204 to (-159.86, 159, -10) mm, rotated rx 180 ry 0 rz 0.01 deg; joints [35.354, -47.27, 106.585, -140.684, 65.995, 162.514] to (-172.35, 157.77, -10) mm, rotated rx -180 ry 0 rz 0.01 deg; joints [35.035, -46.853, 105.716, -140.886, 65.541, 162.34]
  MoveL 205 to (-214.91, 157.56, -10) mm, rotated rx 180 ry 0 rz 0.01 deg; joints [34.104, -45.296, 102.465, -141.355, 63.913, 161.588]
  MoveC 206 to (-237.65, 159.45, -10) mm, rotated rx 180 ry 0 rz 0.01 deg; joints [33.686, -44.388, 100.57, -141.486, 62.998, 161.101] to (-259.75, 165.09, -10) mm, rotated rx 180 ry 0 rz 0.01 deg; joints [33.408, -43.391, 98.487, -141.428, 62.051, 160.477]
  MoveC 207 to (-262.78, 167.3, -10) mm, rotated rx -180 ry 0 rz 0.01 deg; joints [33.414, -43.216, 98.121, -141.358, 61.904, 160.338] to (-264.06, 170.83, -10) mm, rotated rx 180 ry 0 rz 0.01 deg; joints [33.496, -43.077, 97.826, -141.219, 61.812, 160.186]
  MoveC 208 to (-265.25, 174.36, -10) mm, rotated rx 180 ry 0 rz 0.01 deg; joints [33.58, -42.941, 97.536, -141.079, 61.723, 160.034] to (-268.11, 176.74, -10) mm, rotated rx 180 ry 0 rz 0.01 deg; joints [33.595, -42.766, 97.171, -140.998, 61.58, 159.89]
  MoveC 209 to (-273.84, 179.44, -10) mm, rotated rx 180 ry 0 rz 0.01 deg; joints [33.561, -42.469, 96.55, -140.923, 61.316, 159.675] to (-279.42, 182.42, -10) mm, rotated rx 180 ry 0 rz 0.01 deg; joints [33.539, -42.169, 95.922, -140.832, 61.054, 159.451]
  MoveC 210 to (-284.62, 185.58, -10) mm, rotated rx -180 ry 0 rz 0.01 deg; joints [33.531, -41.877, 95.314, -140.73, 60.805, 159.226] to (-289.62, 189.04, -10) mm, rotated rx -180 ry 0 rz 0.01 deg; joints [33.535, -41.584, 94.701, -140.611, 60.559, 158.992]
  MoveC 211 to (-294.48, 192.68, -10) mm, rotated rx 180 ry 0 rz 0.01 deg; joints [33.548, -41.29, 94.086, -140.482, 60.317, 158.75] to (-299.27, 196.43, -10) mm, rotated rx -180 ry 0 rz 0.01 deg; joints [33.565, -40.994, 93.468, -140.347, 60.075, 158.505]
  MoveC 212 to (-301.33, 196.67, -10) mm, rotated rx -180 ry 0 rz 0.01 deg; joints [33.531, -40.903, 93.278, -140.346, 59.986, 158.451] to (-302.43, 194.91, -10) mm, rotated rx 180 ry 0 rz 0.01 deg; joints [33.457, -40.904, 93.283, -140.426, 59.961, 158.494]
  MoveL 213 to (-302.43, 149.11, -10) mm, rotated rx -180 ry 0 rz 0.01 deg; joints [32.074, -42.079, 95.792, -142.379, 60.484, 160.2]
  MoveC 214 to (-301.33, 144.88, -10) mm, rotated rx -180 ry 0 rz 0.01 deg; joints [31.965, -42.229, 96.109, -142.553, 60.577, 160.376] to (-298.32, 141.72, -10) mm, rotated rx 180 ry 0 rz 0.01 deg; joints [31.926, -42.429, 96.53, -142.671, 60.739, 160.551]
  MoveC 215 to (-286.88, 133.71, -10) mm, rotated rx 180 ry 0 rz 0.01 deg; joints [31.899, -43.086, 97.906, -142.941, 61.302, 161.063] to (-276.41, 124.48, -10) mm, rotated rx 180 ry 0 rz 0.01 deg; joints [31.813, -43.725, 99.249, -143.261, 61.836, 161.588]
  MoveC 216 to (-266.95, 114.22, -10) mm, rotated rx -180 ry 0 rz 0.01 deg; joints [31.674, -44.339, 100.545, -143.625, 62.337, 162.118] to (-258.53, 103.09, -10) mm, rotated rx 180 ry 0 rz 0.01 deg; joints [31.484, -44.924, 101.784, -144.028, 62.803, 162.648]
  MoveL 217 to (-242.23, 74.33, -10) mm, rotated rx 180 ry 0 rz 0.01 deg; joints [30.869, -46.194, 104.488, -145.1, 63.78, 163.879]
  MoveC 218 to (-239.12, 71.22, -10) mm, rotated rx -180 ry 0 rz 0.01 deg; joints [30.828, -46.38, 104.882, -145.202, 63.939, 164.032] to (-234.88, 70.09, -10) mm, rotated rx -180 ry 0 rz 0.01 deg; joints [30.874, -46.566, 105.272, -145.21, 64.121, 164.14]
  MoveL 219 to (-158.66, 70.09, -10) mm, rotated rx -180 ry 0 rz 0.01 deg; joints [32.453, -49.35, 111.12, -144.35, 67.075, 165.376]
  MoveC 220 to (-154.41, 71.22, -10) mm, rotated rx -180 ry 0 rz 0.01 deg; joints [32.584, -49.475, 111.382, -144.247, 67.222, 165.408] to (-151.3, 74.33, -10) mm, rotated rx 180 ry 0 rz 0.01 deg; joints [32.758, -49.518, 111.464, -144.075, 67.303, 165.362]
  MoveL 221 to (-138.43, 96.77, -10) mm, rotated rx 180 ry 0 rz 0.01 deg; joints [33.803, -49.474, 111.329, -142.967, 67.521, 164.874]
  MoveC 222 to (-131.45, 107.68, -10) mm, rotated rx 180 ry 0 rz 0.01 deg; joints [34.326, -49.47, 111.3, -142.418, 67.651, 164.645] to (-123.4, 117.82, -10) mm, rotated rx -180 ry 0 rz 0.01 deg; joints [34.848, -49.516, 111.377, -141.886, 67.827, 164.456]
  MoveC 223 to (-110.19, 130.78, -10) mm, rotated rx -180 ry 0 rz 0.01 deg; joints [35.586, -49.666, 111.67, -141.161, 68.155, 164.259] to (-95.22, 141.68, -10) mm, rotated rx 180 ry 0 rz 0.01 deg; joints [36.301, -49.914, 112.172, -140.49, 68.563, 164.153]
  MoveC 224 to (-92.18, 144.87, -10) mm, rotated rx -180 ry 0 rz 0.01 deg; joints [36.479, -49.939, 112.221, -140.313, 68.633, 164.1] to (-91.08, 149.13, -10) mm, rotated rx -180 ry 0 rz 0.01 deg; joints [36.645, -49.875, 112.076, -140.123, 68.622, 163.981]
  MoveL 225 to (-91.08, 194.88, -10) mm, rotated rx -180 ry 0 rz 0.01 deg; joints [38.109, -48.748, 109.623, -138.282, 68.074, 162.481]
  MoveC 226 to (-92.19, 196.64, -10) mm, rotated rx -180 ry 0 rz 0.01 deg; joints [38.137, -48.667, 109.449, -138.228, 68.013, 162.403] to (-94.25, 196.41, -10) mm, rotated rx -180 ry 0 rz 0.01 deg; joints [38.079, -48.603, 109.317, -138.269, 67.943, 162.376]
  MoveC 227 to (-105.38, 188.27, -10) mm, rotated rx 180 ry 0 rz 0.01 deg; joints [37.553, -48.435, 108.976, -138.76, 67.643, 162.462] to (-117.11, 181.04, -10) mm, rotated rx 180 ry 0 rz 0.01 deg; joints [37.043, -48.217, 108.531, -139.22, 67.307, 162.507]
  MoveC 228 to (-129.54, 175.03, -10) mm, rotated rx -180 ry 0 rz 0.01 deg; joints [36.56, -47.939, 107.959, -139.636, 66.927, 162.497] to (-142.62, 170.63, -10) mm, rotated rx 180 ry 0 rz 0.01 deg; joints [36.116, -47.593, 107.241, -139.99, 66.499, 162.421]
  MoveC 229 to (-160.45, 167.02, -10) mm, rotated rx -180 ry 0 rz 0.01 deg; joints [35.594, -47.052, 106.116, -140.363, 65.879, 162.235] to (-178.6, 165.68, -10) mm, rotated rx -180 ry 0 rz 0.01 deg; joints [35.146, -46.434, 104.826, -140.634, 65.213, 161.963]
  MoveL 230 to (-214.91, 165.47, -10) mm, rotated rx 180 ry 0 rz 0.01 deg; joints [34.351, -45.101, 102.044, -141.027, 63.822, 161.314]
  MoveC 231 to (-242.1, 168.32, -10) mm, rotated rx -180 ry 0 rz 0.01 deg; joints [33.869, -43.996, 99.74, -141.153, 62.72, 160.704] to (-268.11, 176.74, -10) mm, rotated rx 180 ry 0 rz 0.01 deg; joints [33.595, -42.766, 97.171, -140.998, 61.58, 159.89]
  MoveC 232 to (-270.85, 179.12, -10) mm, rotated rx 180 ry 0 rz 0.01 deg; joints [33.612, -42.597, 96.815, -140.916, 61.441, 159.748] to (-271.78, 182.63, -10) mm, rotated rx 180 ry 0 rz 0.01 deg; joints [33.699, -42.469, 96.545, -140.775, 61.363, 159.6]
  MoveC 233 to (-272.62, 186.14, -10) mm, rotated rx 180 ry 0 rz 0.01 deg; joints [33.788, -42.345, 96.282, -140.633, 61.289, 159.454] to (-275.18, 188.68, -10) mm, rotated rx -180 ry 0 rz 0.01 deg; joints [33.813, -42.177, 95.929, -140.542, 61.156, 159.307]
  MoveC 234 to (-292.14, 200.05, -10) mm, rotated rx 180 ry 0 rz 0.01 deg; joints [33.814, -41.19, 93.868, -140.157, 60.328, 158.521] to (-307, 214.06, -10) mm, rotated rx 180 ry 0 rz 0.01 deg; joints [33.932, -40.198, 91.794, -139.628, 59.548, 157.651]
  MoveC 235 to (-308.89, 214.52, -10) mm, rotated rx -180 ry 0 rz 0.01 deg; joints [33.909, -40.107, 91.605, -139.615, 59.464, 157.591] to (-309.99, 212.92, -10) mm, rotated rx -180 ry 0 rz 0.01 deg; joints [33.84, -40.104, 91.602, -139.688, 59.436, 157.628]
  MoveL 236 to (-309.99, 144.41, -10) mm, rotated rx -180 ry 0 rz 0.01 deg; joints [31.786, -41.885, 95.398, -142.62, 60.221, 160.216]
  MoveC 237 to (-308.89, 140.36, -10) mm, rotated rx 180 ry 0 rz 0.01 deg; joints [31.682, -42.03, 95.705, -142.787, 60.313, 160.386] to (-305.9, 137.42, -10) mm, rotated rx -180 ry 0 rz 0.01 deg; joints [31.648, -42.225, 96.114, -142.897, 60.471, 160.553]
  MoveC 238 to (-293.97, 129.68, -10) mm, rotated rx -180 ry 0 rz 0.01 deg; joints [31.636, -42.898, 97.523, -143.157, 61.055, 161.067] to (-283.11, 120.5, -10) mm, rotated rx -180 ry 0 rz 0.01 deg; joints [31.558, -43.553, 98.898, -143.477, 61.606, 161.599]
  MoveC 239 to (-273.38, 110.13, -10) mm, rotated rx 180 ry 0 rz 0.01 deg; joints [31.419, -44.181, 100.224, -143.847, 62.121, 162.139] to (-264.77, 98.83, -10) mm, rotated rx 180 ry 0 rz 0.01 deg; joints [31.225, -44.779, 101.489, -144.259, 62.598, 162.679]
  MoveL 240 to (-246.6, 66.78, -10) mm, rotated rx -180 ry 0 rz 0.01 deg; joints [30.534, -46.192, 104.497, -145.46, 63.689, 164.048]
  MoveC 241 to (-243.49, 63.67, -10) mm, rotated rx -180 ry 0 rz 0.01 deg; joints [30.492, -46.378, 104.891, -145.563, 63.848, 164.2] to (-239.25, 62.53, -10) mm, rotated rx -180 ry 0 rz 0.01 deg; joints [30.537, -46.563, 105.282, -145.571, 64.031, 164.307]
  MoveL 242 to (-154.3, 62.53, -10) mm, rotated rx 180 ry 0 rz 0.01 deg; joints [32.289, -49.665, 111.799, -144.61, 67.327, 165.674]
  MoveC 243 to (-150.05, 63.67, -10) mm, rotated rx -180 ry 0 rz 0.01 deg; joints [32.421, -49.79, 112.061, -144.506, 67.473, 165.705] to (-146.94, 66.78, -10) mm, rotated rx -180 ry 0 rz 0.01 deg; joints [32.596, -49.833, 112.144, -144.334, 67.554, 165.66]
  MoveL 244 to (-133.47, 90.53, -10) mm, rotated rx 180 ry 0 rz 0.01 deg; joints [33.704, -49.784, 111.995, -143.157, 67.778, 165.146]
  MoveC 245 to (-126.2, 102.1, -10) mm, rotated rx 180 ry 0 rz 0.01 deg; joints [34.259, -49.777, 111.957, -142.575, 67.91, 164.903] to (-117.73, 112.83, -10) mm, rotated rx 180 ry 0 rz 0.01 deg; joints [34.814, -49.824, 112.036, -142.009, 68.094, 164.703]
  MoveC 246 to (-103.68, 126.37, -10) mm, rotated rx 180 ry 0 rz 0.01 deg; joints [35.594, -49.988, 112.359, -141.244, 68.442, 164.502] to (-87.61, 137.42, -10) mm, rotated rx 180 ry 0 rz 0.01 deg; joints [36.345, -50.268, 112.927, -140.544, 68.886, 164.41]
  MoveC 247 to (-84.62, 140.39, -10) mm, rotated rx 180 ry 0 rz 0.01 deg; joints [36.516, -50.297, 112.984, -140.376, 68.956, 164.363] to (-83.52, 144.46, -10) mm, rotated rx 180 ry 0 rz 0.01 deg; joints [36.676, -50.237, 112.849, -140.193, 68.946, 164.252]
  MoveL 248 to (-83.53, 212.92, -10) mm, rotated rx 180 ry 0 rz 0.01 deg; joints [38.859, -48.537, 109.15, -137.448, 68.124, 161.998]
  MoveC 249 to (-84.63, 214.52, -10) mm, rotated rx 180 ry 0 rz 0.01 deg; joints [38.881, -48.459, 108.983, -137.401, 68.066, 161.924] to (-86.52, 214.08, -10) mm, rotated rx 180 ry 0 rz 0.01 deg; joints [38.82, -48.408, 108.875, -137.448, 68.005, 161.907]
  MoveC 250 to (-96.06, 204.66, -10) mm, rotated rx 180 ry 0 rz 0.01 deg; joints [38.292, -48.332, 108.733, -137.966, 67.78, 162.067] to (-106.49, 196.24, -10) mm, rotated rx 180 ry 0 rz 0.01 deg; joints [37.776, -48.195, 108.46, -138.457, 67.509, 162.175]
  MoveC 251 to (-117.76, 188.97, -10) mm, rotated rx -180 ry 0 rz 0.01 deg; joints [37.277, -47.996, 108.054, -138.91, 67.19, 162.229] to (-129.75, 182.98, -10) mm, rotated rx -180 ry 0 rz 0.01 deg; joints [36.805, -47.733, 107.514, -139.317, 66.825, 162.226]
  MoveC 252 to (-150.35, 176.31, -10) mm, rotated rx 180 ry 0 rz 0.01 deg; joints [36.117, -47.18, 106.368, -139.858, 66.147, 162.096] to (-171.82, 173.64, -10) mm, rotated rx 180 ry 0 rz 0.01 deg; joints [35.547, -46.482, 104.911, -140.229, 65.376, 161.811]
  MoveL 253 to (-214.91, 173.03, -10) mm, rotated rx 180 ry 0 rz 0.01 deg; joints [34.586, -44.913, 101.639, -140.714, 63.734, 161.051]
  MoveC 254 to (-246.04, 177.01, -10) mm, rotated rx 180 ry 0 rz 0.01 deg; joints [34.054, -43.625, 98.953, -140.823, 62.463, 160.317] to (-275.18, 188.68, -10) mm, rotated rx 180 ry 0 rz 0.01 deg; joints [33.813, -42.177, 95.929, -140.542, 61.156, 159.307]
  MoveC 255 to (-277.57, 191.16, -10) mm, rotated rx 180 ry 0 rz 0.01 deg; joints [33.84, -42.016, 95.592, -140.452, 61.03, 159.165] to (-278.16, 194.55, -10) mm, rotated rx -180 ry 0 rz 0.01 deg; joints [33.929, -41.903, 95.353, -140.312, 60.966, 159.026]
  MoveC 256 to (-278.7, 197.94, -10) mm, rotated rx -180 ry 0 rz 0.01 deg; joints [34.02, -41.793, 95.118, -140.172, 60.905, 158.888] to (-280.93, 200.53, -10) mm, rotated rx -180 ry 0 rz 0.01 deg; joints [34.052, -41.634, 94.785, -140.076, 60.784, 158.743]
  MoveC 257 to (-286.58, 204.46, -10) mm, rotated rx -180 ry 0 rz 0.01 deg; joints [34.056, -41.3, 94.088, -139.941, 60.507, 158.473] to (-292.01, 208.68, -10) mm, rotated rx 180 ry 0 rz 0.01 deg; joints [34.072, -40.965, 93.388, -139.79, 60.234, 158.194]
  MoveC 258 to (-298.39, 214.58, -10) mm, rotated rx 180 ry 0 rz 0.01 deg; joints [34.118, -40.542, 92.504, -139.569, 59.902, 157.825] to (-304.04, 221.18, -10) mm, rotated rx -180 ry 0 rz 0.01 deg; joints [34.199, -40.126, 91.635, -139.311, 59.59, 157.439]
  MoveC 259 to (-309.2, 228.15, -10) mm, rotated rx 180 ry 0 rz 0.01 deg; joints [34.3, -39.716, 90.778, -139.032, 59.292, 157.044] to (-314.21, 235.23, -10) mm, rotated rx -180 ry 0 rz 0.01 deg; joints [34.405, -39.306, 89.919, -138.744, 58.999, 156.643]
  MoveC 260 to (-315.96, 235.84, -10) mm, rotated rx -180 ry 0 rz 0.01 deg; joints [34.388, -39.214, 89.73, -138.723, 58.918, 156.577] to (-317.06, 234.34, -10) mm, rotated rx 180 ry 0 rz 0.01 deg; joints [34.324, -39.21, 89.723, -138.791, 58.889, 156.611]
  MoveL 261 to (-317.06, 140.03, -10) mm, rotated rx 180 ry 0 rz 0.01 deg; joints [31.517, -41.701, 95.024, -142.842, 59.973, 160.231]
  MoveC 262 to (-315.92, 135.98, -10) mm, rotated rx 180 ry 0 rz 0.01 deg; joints [31.414, -41.848, 95.334, -143.01, 60.066, 160.401] to (-312.84, 133.12, -10) mm, rotated rx 180 ry 0 rz 0.01 deg; joints [31.384, -42.045, 95.747, -143.117, 60.228, 160.567]
  MoveC 263 to (-300.79, 125.89, -10) mm, rotated rx -180 ry 0 rz 0.01 deg; joints [31.388, -42.713, 97.145, -143.36, 60.814, 161.067] to (-289.79, 117.13, -10) mm, rotated rx -180 ry 0 rz 0.01 deg; joints [31.324, -43.365, 98.514, -143.664, 61.369, 161.588]
  MoveC 264 to (-279.97, 107.09, -10) mm, rotated rx -180 ry 0 rz 0.01 deg; joints [31.194, -43.991, 99.834, -144.024, 61.886, 162.12] to (-271.38, 95.97, -10) mm, rotated rx 180 ry 0 rz 0.01 deg; joints [31.005, -44.585, 101.09, -144.431, 62.361, 162.655]
  MoveL 265 to (-250.66, 59.68, -10) mm, rotated rx 180 ry 0 rz 0.01 deg; joints [30.22, -46.189, 104.504, -145.797, 63.604, 164.206]
  MoveC 266 to (-247.58, 56.59, -10) mm, rotated rx 180 ry 0 rz 0.01 deg; joints [30.177, -46.373, 104.895, -145.9, 63.763, 164.356] to (-243.37, 55.46, -10) mm, rotated rx -180 ry 0 rz 0.01 deg; joints [30.221, -46.558, 105.283, -145.909, 63.944, 164.462]
  MoveL 267 to (-150.14, 55.46, -10) mm, rotated rx -180 ry 0 rz 0.01 deg; joints [32.136, -49.961, 112.437, -144.852, 67.565, 165.951]
  MoveC 268 to (-145.96, 56.58, -10) mm, rotated rx 180 ry 0 rz 0.01 deg; joints [32.266, -50.084, 112.694, -144.748, 67.709, 165.981] to (-142.9, 59.64, -10) mm, rotated rx 180 ry 0 rz 0.01 deg; joints [32.438, -50.126, 112.777, -144.578, 67.788, 165.937]
  MoveL 269 to (-124.32, 91.78, -10) mm, rotated rx -180 ry 0 rz 0.01 deg; joints [33.954, -50.071, 112.599, -142.975, 68.101, 165.251]
  MoveC 270 to (-113.01, 107.84, -10) mm, rotated rx 180 ry 0 rz 0.01 deg; joints [34.756, -50.098, 112.624, -142.145, 68.325, 164.934] to (-99.01, 121.62, -10) mm, rotated rx -180 ry 0 rz 0.01 deg; joints [35.547, -50.256, 112.931, -141.367, 68.667, 164.726]
  MoveC 271 to (-94.69, 124.91, -10) mm, rotated rx 180 ry 0 rz 0.01 deg; joints [35.76, -50.324, 113.07, -141.166, 68.783, 164.691] to (-90.14, 127.87, -10) mm, rotated rx 180 ry 0 rz 0.01 deg; joints [35.968, -50.407, 113.239, -140.973, 68.91, 164.67]
  MoveC 272 to (-85.44, 130.59, -10) mm, rotated rx -180 ry 0 rz 0.01 deg; joints [36.172, -50.5, 113.43, -140.788, 69.045, 164.659] to (-80.66, 133.15, -10) mm, rotated rx 180 ry 0 rz 0.01 deg; joints [36.373, -50.598, 113.634, -140.607, 69.184, 164.655]
  MoveC 273 to (-77.59, 136, -10) mm, rotated rx -180 ry 0 rz 0.01 deg; joints [36.543, -50.632, 113.701, -140.441, 69.258, 164.614] to (-76.46, 140.03, -10) mm, rotated rx 180 ry 0 rz 0.01 deg; joints [36.704, -50.575, 113.572, -140.259, 69.25, 164.504]
  MoveL 274 to (-76.46, 234.32, -10) mm, rotated rx -180 ry 0 rz 0.01 deg; joints [39.693, -48.209, 108.426, -136.493, 68.116, 161.382]
  MoveC 275 to (-77.55, 235.81, -10) mm, rotated rx 180 ry 0 rz 0.01 deg; joints [39.71, -48.134, 108.264, -136.452, 68.06, 161.312] to (-79.3, 235.2, -10) mm, rotated rx -180 ry 0 rz 0.01 deg; joints [39.648, -48.092, 108.178, -136.502, 68.006, 161.303]
  MoveL 276 to (-85.77, 225.74, -10) mm, rotated rx -180 ry 0 rz 0.01 deg; joints [39.197, -48.128, 108.269, -136.974, 67.892, 161.52]
  MoveC 277 to (-89.21, 221.09, -10) mm, rotated rx 180 ry 0 rz 0.01 deg; joints [38.969, -48.135, 108.292, -137.21, 67.827, 161.621] to (-92.98, 216.71, -10) mm, rotated rx 180 ry 0 rz 0.01 deg; joints [38.741, -48.123, 108.275, -137.441, 67.745, 161.707]
  MoveC 278 to (-110.06, 201.79, -10) mm, rotated rx -180 ry 0 rz 0.01 deg; joints [37.862, -47.932, 107.899, -138.286, 67.314, 161.926] to (-129.86, 190.72, -10) mm, rotated rx -180 ry 0 rz 0.01 deg; joints [37.045, -47.535, 107.085, -139.006, 66.73, 161.962]
  MoveC 279 to (-151.35, 183.6, -10) mm, rotated rx -180 ry 0 rz 0.01 deg; joints [36.323, -46.963, 105.9, -139.575, 66.024, 161.831] to (-173.74, 180.26, -10) mm, rotated rx 180 ry 0 rz 0.01 deg; joints [35.711, -46.247, 104.409, -139.98, 65.226, 161.55]
  MoveL 280 to (-214.91, 180.1, -10) mm, rotated rx 180 ry 0 rz 0.01 deg; joints [34.804, -44.735, 101.257, -140.421, 63.653, 160.802]
  MoveC 281 to (-235.77, 182.01, -10) mm, rotated rx 180 ry 0 rz 0.01 deg; joints [34.421, -43.894, 99.504, -140.53, 62.813, 160.337] to (-255.94, 187.7, -10) mm, rotated rx -180 ry 0 rz 0.01 deg; joints [34.175, -42.965, 97.566, -140.452, 61.945, 159.735]
  MoveC 282 to (-268.78, 193.44, -10) mm, rotated rx 180 ry 0 rz 0.01 deg; joints [34.086, -42.308, 96.193, -140.3, 61.361, 159.262] to (-280.93, 200.53, -10) mm, rotated rx 180 ry 0 rz 0.01 deg; joints [34.052, -41.634, 94.785, -140.076, 60.784, 158.743]
  MoveC 283 to (-282.97, 203, -10) mm, rotated rx 180 ry 0 rz 0.01 deg; joints [34.084, -41.485, 94.474, -139.983, 60.672, 158.606] to (-283.28, 206.19, -10) mm, rotated rx 180 ry 0 rz 0.01 deg; joints [34.173, -41.388, 94.267, -139.85, 60.623, 158.478]
  MoveC 284 to (-283.52, 209.36, -10) mm, rotated rx -180 ry 0 rz 0.01 deg; joints [34.262, -41.293, 94.066, -139.717, 60.576, 158.352] to (-285.39, 211.94, -10) mm, rotated rx 180 ry 0 rz 0.01 deg; joints [34.301, -41.147, 93.76, -139.618, 60.469, 158.213]
  MoveC 285 to (-286.59, 212.88, -10) mm, rotated rx -180 ry 0 rz 0.01 deg; joints [34.304, -41.073, 93.605, -139.584, 60.409, 158.151] to (-287.77, 213.84, -10) mm, rotated rx 180 ry 0 rz 0.01 deg; joints [34.309, -40.999, 93.45, -139.55, 60.349, 158.088]
  MoveC 286 to (-297.45, 223, -10) mm, rotated rx 180 ry 0 rz 0.01 deg; joints [34.383, -40.35, 92.095, -139.206, 59.843, 157.517] to (-305.74, 233.42, -10) mm, rotated rx -180 ry 0 rz 0.01 deg; joints [34.521, -39.714, 90.765, -138.794, 59.376, 156.914]
  MoveC 287 to (-312.64, 244.8, -10) mm, rotated rx 180 ry 0 rz 0.01 deg; joints [34.711, -39.1, 89.48, -138.328, 58.953, 156.292] to (-318.26, 256.87, -10) mm, rotated rx -180 ry 0 rz 0.01 deg; joints [34.944, -38.511, 88.247, -137.821, 58.574, 155.659]
  MoveC 288 to (-321.43, 258.6, -10) mm, rotated rx -180 ry 0 rz 0.01 deg; joints [34.93, -38.323, 87.859, -137.752, 58.419, 155.508] to (-323.73, 255.81, -10) mm, rotated rx -180 ry 0 rz 0.01 deg; joints [34.806, -38.306, 87.826, -137.878, 58.354, 155.567]
  MoveL 289 to (-323.73, 135.95, -10) mm, rotated rx -180 ry 0 rz 0.01 deg; joints [31.267, -41.524, 94.663, -143.048, 59.736, 160.241]
  MoveC 290 to (-322.59, 131.91, -10) mm, rotated rx -180 ry 0 rz 0.01 deg; joints [31.164, -41.67, 94.973, -143.216, 59.83, 160.412] to (-319.52, 129.05, -10) mm, rotated rx 180 ry 0 rz 0.01 deg; joints [31.133, -41.867, 95.386, -143.324, 59.992, 160.578]
  MoveC 291 to (-315.45, 126.98, -10) mm, rotated rx 180 ry 0 rz 0.01 deg; joints [31.145, -42.086, 95.843, -143.393, 60.187, 160.735] to (-311.37, 124.93, -10) mm, rotated rx -180 ry 0 rz 0.01 deg; joints [31.158, -42.303, 96.297, -143.46, 60.382, 160.891]
  MoveC 292 to (-307.36, 122.73, -10) mm, rotated rx 180 ry 0 rz 0.01 deg; joints [31.165, -42.52, 96.75, -143.532, 60.575, 161.049] to (-303.55, 120.22, -10) mm, rotated rx 180 ry 0 rz 0.01 deg; joints [31.159, -42.736, 97.202, -143.618, 60.763, 161.213]
  MoveC 293 to (-295.7, 113.93, -10) mm, rotated rx -180 ry 0 rz 0.01 deg; joints [31.11, -43.202, 98.182, -143.839, 61.16, 161.586] to (-288.56, 106.84, -10) mm, rotated rx -180 ry 0 rz 0.01 deg; joints [31.022, -43.655, 99.134, -144.094, 61.535, 161.968]
  MoveC 294 to (-282.07, 99.17, -10) mm, rotated rx -180 ry 0 rz 0.01 deg; joints [30.902, -44.09, 100.054, -144.375, 61.888, 162.351] to (-276.12, 91.07, -10) mm, rotated rx -180 ry 0 rz 0.01 deg; joints [30.756, -44.51, 100.942, -144.675, 62.222, 162.734]
  MoveL 295 to (-254.45, 52.85, -10) mm, rotated rx -180 ry 0 rz 0.01 deg; joints [29.921, -46.19, 104.518, -146.12, 63.527, 164.36]
  MoveC 296 to (-251.56, 49.88, -10) mm, rotated rx 180 ry 0 rz 0.01 deg; joints [29.877, -46.363, 104.886, -146.221, 63.677, 164.502] to (-247.56, 48.79, -10) mm, rotated rx 180 ry 0 rz 0.01 deg; joints [29.918, -46.539, 105.257, -146.231, 63.85, 164.603]
  MoveL 297 to (-145.88, 48.79, -10) mm, rotated rx -180 ry 0 rz 0.01 deg; joints [31.997, -50.25, 113.06, -145.075, 67.802, 166.215]
  MoveC 298 to (-141.92, 49.88, -10) mm, rotated rx -180 ry 0 rz 0.01 deg; joints [32.122, -50.365, 113.302, -144.975, 67.938, 166.243] to (-139.08, 52.85, -10) mm, rotated rx 180 ry 0 rz 0.01 deg; joints [32.287, -50.401, 113.374, -144.811, 68.01, 166.198]
  MoveC 299 to (-129.5, 70.17, -10) mm, rotated rx -180 ry 0 rz 0.01 deg; joints [33.099, -50.365, 113.262, -143.95, 68.164, 165.827] to (-119.55, 87.28, -10) mm, rotated rx 180 ry 0 rz 0.01 deg; joints [33.91, -50.334, 113.162, -143.093, 68.329, 165.463]
  MoveC 300 to (-107.95, 103.41, -10) mm, rotated rx 180 ry 0 rz 0.01 deg; joints [34.725, -50.369, 113.205, -142.253, 68.561, 165.15] to (-93.75, 117.3, -10) mm, rotated rx -180 ry 0 rz 0.01 deg; joints [35.528, -50.531, 113.521, -141.463, 68.908, 164.943]
  MoveC 301 to (-89.12, 120.74, -10) mm, rotated rx 180 ry 0 rz 0.01 deg; joints [35.754, -50.606, 113.673, -141.249, 69.032, 164.909] to (-84.19, 123.71, -10) mm, rotated rx 180 ry 0 rz 0.01 deg; joints [35.973, -50.701, 113.869, -141.049, 69.172, 164.894]
  MoveC 302 to (-79.11, 126.41, -10) mm, rotated rx -180 ry 0 rz 0.01 deg; joints [36.187, -50.806, 114.086, -140.856, 69.32, 164.89] to (-74, 129.06, -10) mm, rotated rx -180 ry 0 rz 0.01 deg; joints [36.4, -50.913, 114.307, -140.665, 69.469, 164.888]
  MoveC 303 to (-70.92, 131.91, -10) mm, rotated rx 180 ry 0 rz 0.01 deg; joints [36.571, -50.947, 114.374, -140.498, 69.543, 164.847] to (-69.78, 135.94, -10) mm, rotated rx -180 ry 0 rz 0.01 deg; joints [36.733, -50.89, 114.245, -140.315, 69.534, 164.739]
  MoveL 304 to (-69.79, 255.8, -10) mm, rotated rx -180 ry 0 rz 0.01 deg; joints [40.509, -47.851, 107.639, -135.548, 68.091, 160.745]
  MoveC 305 to (-72.09, 258.59, -10) mm, rotated rx -180 ry 0 rz 0.01 deg; joints [40.534, -47.699, 107.316, -135.475, 67.978, 160.606] to (-75.26, 256.85, -10) mm, rotated rx 180 ry 0 rz 0.01 deg; joints [40.402, -47.642, 107.199, -135.592, 67.888, 160.613]
  MoveC 306 to (-85.39, 237.38, -10) mm, rotated rx 180 ry 0 rz 0.01 deg; joints [39.561, -47.832, 107.629, -136.51, 67.767, 161.122] to (-99.16, 220.28, -10) mm, rotated rx -180 ry 0 rz 0.01 deg; joints [38.699, -47.823, 107.638, -137.39, 67.484, 161.479]
  MoveC 307 to (-115.99, 206.2, -10) mm, rotated rx 180 ry 0 rz 0.01 deg; joints [37.856, -47.617, 107.231, -138.193, 67.049, 161.673] to (-135.21, 195.59, -10) mm, rotated rx 180 ry 0 rz 0.01 deg; joints [37.071, -47.225, 106.429, -138.881, 66.477, 161.703]
  MoveC 308 to (-154.49, 189.41, -10) mm, rotated rx 180 ry 0 rz 0.01 deg; joints [36.432, -46.705, 105.35, -139.378, 65.839, 161.577] to (-174.61, 187.1, -10) mm, rotated rx 180 ry 0 rz 0.01 deg; joints [35.904, -46.043, 103.972, -139.711, 65.114, 161.298]
  MoveL 309 to (-214.91, 186.77, -10) mm, rotated rx -180 ry 0 rz 0.01 deg; joints [35.009, -44.566, 100.893, -140.146, 63.575, 160.566]
  MoveC 310 to (-234.63, 188.59, -10) mm, rotated rx -180 ry 0 rz 0.01 deg; joints [34.645, -43.769, 99.234, -140.247, 62.782, 160.123] to (-253.69, 193.98, -10) mm, rotated rx -180 ry 0 rz 0.01 deg; joints [34.412, -42.89, 97.4, -140.172, 61.963, 159.55]
  MoveC 311 to (-270.2, 201.79, -10) mm, rotated rx 180 ry 0 rz 0.01 deg; joints [34.307, -42.032, 95.607, -139.958, 61.207, 158.921] to (-285.39, 211.94, -10) mm, rotated rx -180 ry 0 rz 0.01 deg; joints [34.301, -41.147, 93.76, -139.618, 60.469, 158.213]
  MoveC 312 to (-288, 215.68, -10) mm, rotated rx -180 ry 0 rz 0.01 deg; joints [34.358, -40.939, 93.324, -139.473, 60.318, 158.012] to (-288.03, 220.25, -10) mm, rotated rx -180 ry 0 rz 0.01 deg; joints [34.492, -40.814, 93.057, -139.279, 60.264, 157.834]
  MoveC 313 to (-287.9, 224.76, -10) mm, rotated rx -180 ry 0 rz 0.01 deg; joints [34.627, -40.695, 92.805, -139.087, 60.217, 157.662] to (-290.04, 228.73, -10) mm, rotated rx 180 ry 0 rz 0.01 deg; joints [34.699, -40.498, 92.39, -138.929, 60.083, 157.459]
  MoveC 314 to (-295.05, 234.52, -10) mm, rotated rx 180 ry 0 rz 0.01 deg; joints [34.767, -40.129, 91.62, -138.704, 59.808, 157.117] to (-299.55, 240.73, -10) mm, rotated rx 180 ry 0 rz 0.01 deg; joints [34.856, -39.767, 90.863, -138.458, 59.549, 156.766]
  MoveC 315 to (-306.11, 252.25, -10) mm, rotated rx -180 ry 0 rz 0.01 deg; joints [35.055, -39.162, 89.597, -137.987, 59.14, 156.145] to (-311.1, 264.54, -10) mm, rotated rx -180 ry 0 rz 0.01 deg; joints [35.304, -38.592, 88.403, -137.472, 58.785, 155.517]
  MoveC 316 to (-313.2, 267.41, -10) mm, rotated rx 180 ry 0 rz 0.01 deg; joints [35.343, -38.417, 88.038, -137.353, 58.663, 155.345] to (-316.59, 268.51, -10) mm, rotated rx 180 ry 0 rz 0.01 deg; joints [35.306, -38.239, 87.67, -137.313, 58.506, 155.214]
  MoveL 317 to (-329.24, 268.51, -10) mm, rotated rx 180 ry 0 rz 0.01 deg; joints [35.055, -37.69, 86.54, -137.333, 57.968, 154.893]
  MoveC 318 to (-331.97, 267.38, -10) mm, rotated rx -180 ry 0 rz 0.01 deg; joints [34.97, -37.604, 86.365, -137.386, 57.864, 154.87] to (-333.09, 264.66, -10) mm, rotated rx 180 ry 0 rz 0.01 deg; joints [34.872, -37.636, 86.435, -137.506, 57.848, 154.957]
  MoveL 319 to (-333.09, 129.75, -10) mm, rotated rx -180 ry 0 rz 0.01 deg; joints [30.903, -41.283, 94.175, -143.354, 59.407, 160.272]
  MoveC 320 to (-332, 125.98, -10) mm, rotated rx 180 ry 0 rz 0.01 deg; joints [30.807, -41.421, 94.466, -143.512, 59.496, 160.432] to (-329.06, 123.38, -10) mm, rotated rx -180 ry 0 rz 0.01 deg; joints [30.781, -41.606, 94.855, -143.612, 59.65, 160.587]
  MoveC 321 to (-321.21, 119.46, -10) mm, rotated rx -180 ry 0 rz 0.01 deg; joints [30.804, -42.028, 95.735, -143.744, 60.028, 160.889] to (-313.53, 115.19, -10) mm, rotated rx -180 ry 0 rz 0.01 deg; joints [30.814, -42.446, 96.61, -143.888, 60.4, 161.194]
  MoveC 322 to (-306.22, 110.3, -10) mm, rotated rx 180 ry 0 rz 0.01 deg; joints [30.798, -42.861, 97.479, -144.057, 60.761, 161.509] to (-299.56, 104.57, -10) mm, rotated rx 180 ry 0 rz 0.01 deg; joints [30.742, -43.265, 98.329, -144.261, 61.104, 161.838]
  MoveC 323 to (-288.54, 92.19, -10) mm, rotated rx -180 ry 0 rz 0.01 deg; joints [30.556, -43.992, 99.862, -144.717, 61.699, 162.469] to (-279.43, 78.34, -10) mm, rotated rx -180 ry 0 rz 0.01 deg; joints [30.282, -44.664, 101.286, -145.241, 62.228, 163.099]
  MoveL 324 to (-263.11, 49.58, -10) mm, rotated rx 180 ry 0 rz 0.01 deg; joints [29.647, -45.924, 103.969, -146.334, 63.212, 164.318]
  MoveC 325 to (-262.3, 48.09, -10) mm, rotated rx -180 ry 0 rz 0.01 deg; joints [29.613, -45.987, 104.104, -146.391, 63.261, 164.379] to (-261.57, 46.55, -10) mm, rotated rx -180 ry 0 rz 0.01 deg; joints [29.575, -46.048, 104.233, -146.45, 63.307, 164.44]
  MoveC 326 to (-260.88, 44.99, -10) mm, rotated rx -180 ry 0 rz 0.01 deg; joints [29.537, -46.107, 104.36, -146.51, 63.353, 164.501] to (-260.18, 43.44, -10) mm, rotated rx 180 ry 0 rz 0.01 deg; joints [29.498, -46.167, 104.488, -146.57, 63.398, 164.562]
  MoveC 327 to (-257.63, 40.52, -10) mm, rotated rx 180 ry 0 rz 0.01 deg; joints [29.448, -46.326, 104.827, -146.673, 63.534, 164.697] to (-253.9, 39.42, -10) mm, rotated rx 180 ry 0 rz 0.01 deg; joints [29.482, -46.492, 105.176, -146.686, 63.697, 164.793]
  MoveL 328 to (-139.65, 39.42, -10) mm, rotated rx -180 ry 0 rz 0.01 deg; joints [31.806, -50.66, 113.948, -145.385, 68.145, 166.585]
  MoveC 329 to (-135.89, 40.52, -10) mm, rotated rx 180 ry 0 rz 0.01 deg; joints [31.926, -50.768, 114.174, -145.286, 68.273, 166.61] to (-133.3, 43.45, -10) mm, rotated rx -180 ry 0 rz 0.01 deg; joints [32.086, -50.797, 114.23, -145.126, 68.335, 166.563]
  MoveC 330 to (-132.49, 45.2, -10) mm, rotated rx 180 ry 0 rz 0.01 deg; joints [32.165, -50.789, 114.209, -145.041, 68.345, 166.524] to (-131.72, 46.96, -10) mm, rotated rx 180 ry 0 rz 0.01 deg; joints [32.244, -50.779, 114.184, -144.956, 68.353, 166.484]
  MoveC 331 to (-130.91, 48.71, -10) mm, rotated rx 180 ry 0 rz 0.01 deg; joints [32.323, -50.77, 114.163, -144.87, 68.363, 166.444] to (-130, 50.41, -10) mm, rotated rx -180 ry 0 rz 0.01 deg; joints [32.403, -50.766, 114.151, -144.786, 68.377, 166.408]
  MoveL 332 to (-108.96, 86.15, -10) mm, rotated rx 180 ry 0 rz 0.01 deg; joints [34.116, -50.718, 113.978, -142.982, 68.73, 165.662]
  MoveC 333 to (-96.19, 102.68, -10) mm, rotated rx 180 ry 0 rz 0.01 deg; joints [34.978, -50.781, 114.078, -142.102, 68.995, 165.356] to (-79.89, 115.74, -10) mm, rotated rx -180 ry 0 rz 0.01 deg; joints [35.81, -51.026, 114.573, -141.306, 69.421, 165.209]
  MoveC 334 to (-76.15, 117.89, -10) mm, rotated rx -180 ry 0 rz 0.01 deg; joints [35.973, -51.1, 114.725, -141.156, 69.528, 165.201] to (-72.28, 119.78, -10) mm, rotated rx 180 ry 0 rz 0.01 deg; joints [36.132, -51.184, 114.898, -141.015, 69.642, 165.202]
  MoveC 335 to (-68.35, 121.56, -10) mm, rotated rx -180 ry 0 rz 0.01 deg; joints [36.288, -51.271, 115.08, -140.877, 69.759, 165.209] to (-64.44, 123.39, -10) mm, rotated rx -180 ry 0 rz 0.01 deg; joints [36.446, -51.356, 115.257, -140.736, 69.874, 165.213]
  MoveC 336 to (-61.51, 125.98, -10) mm, rotated rx -180 ry 0 rz 0.01 deg; joints [36.606, -51.391, 115.327, -140.581, 69.946, 165.178] to (-60.42, 129.74, -10) mm, rotated rx -180 ry 0 rz 0.01 deg; joints [36.759, -51.339, 115.209, -140.409, 69.938, 165.079]
  MoveL 337 to (-60.42, 264.66, -10) mm, rotated rx 180 ry 0 rz 0.01 deg; joints [41.014, -47.914, 107.757, -135.056, 68.309, 160.593]
  MoveC 338 to (-61.55, 267.39, -10) mm, rotated rx 180 ry 0 rz 0.01 deg; joints [41.065, -47.802, 107.518, -134.968, 68.237, 160.476] to (-64.28, 268.52, -10) mm, rotated rx -180 ry 0 rz 0.01 deg; joints [41.028, -47.682, 107.265, -134.967, 68.13, 160.389]
  MoveL 339 to (-76.92, 268.52, -10) mm, rotated rx 180 ry 0 rz 0.01 deg; joints [40.706, -47.266, 106.394, -135.162, 67.692, 160.168]
  MoveC 340 to (-80.31, 267.42, -10) mm, rotated rx -180 ry 0 rz 0.01 deg; joints [40.587, -47.184, 106.224, -135.256, 67.587, 160.148] to (-82.41, 264.54, -10) mm, rotated rx -180 ry 0 rz 0.01 deg; joints [40.449, -47.193, 106.248, -135.399, 67.547, 160.213]
  MoveC 341 to (-91.29, 245.22, -10) mm, rotated rx -180 ry 0 rz 0.01 deg; joints [39.65, -47.424, 106.763, -136.289, 67.465, 160.745] to (-104.21, 228.32, -10) mm, rotated rx 180 ry 0 rz 0.01 deg; joints [38.82, -47.44, 106.824, -137.144, 67.208, 161.112]
  MoveC 342 to (-120.36, 214.52, -10) mm, rotated rx -180 ry 0 rz 0.01 deg; joints [38.007, -47.252, 106.452, -137.921, 66.793, 161.31] to (-138.92, 204.19, -10) mm, rotated rx -180 ry 0 rz 0.01 deg; joints [37.25, -46.876, 105.682, -138.583, 66.24, 161.342]
  MoveC 343 to (-157.31, 198.34, -10) mm, rotated rx 180 ry 0 rz 0.01 deg; joints [36.643, -46.377, 104.65, -139.05, 65.629, 161.218] to (-176.5, 196.27, -10) mm, rotated rx -180 ry 0 rz 0.01 deg; joints [36.144, -45.741, 103.326, -139.358, 64.935, 160.944]
  MoveL 344 to (-214.91, 196.13, -10) mm, rotated rx 180 ry 0 rz 0.01 deg; joints [35.295, -44.325, 100.377, -139.759, 63.467, 160.232]
  MoveC 345 to (-233.03, 197.81, -10) mm, rotated rx -180 ry 0 rz 0.01 deg; joints [34.959, -43.592, 98.851, -139.85, 62.739, 159.82] to (-250.53, 202.8, -10) mm, rotated rx 180 ry 0 rz 0.01 deg; joints [34.742, -42.783, 97.163, -139.781, 61.987, 159.288]
  MoveC 346 to (-266.91, 210.69, -10) mm, rotated rx 180 ry 0 rz 0.01 deg; joints [34.639, -41.926, 95.374, -139.563, 61.237, 158.655] to (-281.83, 221.08, -10) mm, rotated rx 180 ry 0 rz 0.01 deg; joints [34.642, -41.044, 93.532, -139.212, 60.509, 157.939]
  MoveC 347 to (-286.06, 224.77, -10) mm, rotated rx -180 ry 0 rz 0.01 deg; joints [34.664, -40.77, 92.96, -139.077, 60.293, 157.702] to (-290.04, 228.73, -10) mm, rotated rx 180 ry 0 rz 0.01 deg; joints [34.699, -40.498, 92.39, -138.929, 60.083, 157.459]
  MoveC 348 to (-292.05, 232.85, -10) mm, rotated rx -180 ry 0 rz 0.01 deg; joints [34.779, -40.3, 91.976, -138.763, 59.952, 157.251] to (-291.37, 237.39, -10) mm, rotated rx -180 ry 0 rz 0.01 deg; joints [34.924, -40.201, 91.765, -138.567, 59.927, 157.087]
  MoveC 349 to (-290.5, 241.83, -10) mm, rotated rx -180 ry 0 rz 0.01 deg; joints [35.07, -40.112, 91.573, -138.374, 59.911, 156.931] to (-291.95, 246.12, -10) mm, rotated rx 180 ry 0 rz 0.01 deg; joints [35.164, -39.93, 91.192, -138.197, 59.801, 156.726]
  MoveC 350 to (-292.81, 247.45, -10) mm, rotated rx -180 ry 0 rz 0.01 deg; joints [35.185, -39.857, 91.039, -138.144, 59.75, 156.653] to (-293.64, 248.78, -10) mm, rotated rx 180 ry 0 rz 0.01 deg; joints [35.207, -39.784, 90.886, -138.091, 59.7, 156.58]
  MoveC 351 to (-299.77, 260.91, -10) mm, rotated rx 180 ry 0 rz 0.01 deg; joints [35.429, -39.178, 89.617, -137.595, 59.303, 155.943] to (-303.97, 273.83, -10) mm, rotated rx -180 ry 0 rz 0.01 deg; joints [35.709, -38.62, 88.447, -137.053, 58.975, 155.306]
  MoveC 352 to (-305.84, 276.74, -10) mm, rotated rx 180 ry 0 rz 0.01 deg; joints [35.753, -38.454, 88.1, -136.933, 58.862, 155.137] to (-309.11, 277.87, -10) mm, rotated rx 180 ry 0 rz 0.01 deg; joints [35.719, -38.28, 87.741, -136.892, 58.711, 155.008]
  MoveL 353 to (-338.6, 277.87, -10) mm, rotated rx -180 ry 0 rz 0.01 deg; joints [35.133, -36.994, 85.094, -136.929, 57.453, 154.245]
  MoveC 354 to (-341.33, 276.74, -10) mm, rotated rx -180 ry 0 rz 0.01 deg; joints [35.049, -36.907, 84.917, -136.979, 57.349, 154.221] to (-342.46, 274.02, -10) mm, rotated rx -180 ry 0 rz 0.01 deg; joints [34.951, -36.94, 84.988, -137.099, 57.333, 154.309]
  MoveL 355 to (-342.45, 123.09, -10) mm, rotated rx -180 ry 0 rz 0.01 deg; joints [30.527, -41.049, 93.701, -143.678, 59.079, 160.319]
  MoveC 356 to (-341.36, 119.56, -10) mm, rotated rx -180 ry 0 rz 0.01 deg; joints [30.438, -41.18, 93.979, -143.826, 59.165, 160.471] to (-338.48, 117.25, -10) mm, rotated rx 180 ry 0 rz 0.01 deg; joints [30.419, -41.358, 94.351, -143.915, 59.315, 160.615]
  MoveC 357 to (-329.76, 113.48, -10) mm, rotated rx -180 ry 0 rz 0.01 deg; joints [30.461, -41.814, 95.302, -144.041, 59.731, 160.929] to (-321.32, 109.16, -10) mm, rotated rx -180 ry 0 rz 0.01 deg; joints [30.481, -42.268, 96.25, -144.187, 60.138, 161.253]
  MoveC 358 to (-313.32, 104.01, -10) mm, rotated rx -180 ry 0 rz 0.01 deg; joints [30.467, -42.717, 97.192, -144.366, 60.533, 161.592] to (-306.08, 97.85, -10) mm, rotated rx 180 ry 0 rz 0.01 deg; joints [30.407, -43.156, 98.113, -144.588, 60.906, 161.945]
  MoveC 359 to (-295.49, 85.95, -10) mm, rotated rx 180 ry 0 rz 0.01 deg; joints [30.225, -43.854, 99.587, -145.03, 61.479, 162.552] to (-286.75, 72.63, -10) mm, rotated rx 180 ry 0 rz 0.01 deg; joints [29.959, -44.5, 100.955, -145.537, 61.989, 163.157]
  MoveL 360 to (-271.09, 44.99, -10) mm, rotated rx -180 ry 0 rz 0.01 deg; joints [29.345, -45.711, 103.532, -146.596, 62.936, 164.33]
  MoveC 361 to (-269.72, 42.39, -10) mm, rotated rx 180 ry 0 rz 0.01 deg; joints [29.284, -45.819, 103.762, -146.695, 63.021, 164.435] to (-268.56, 39.69, -10) mm, rotated rx 180 ry 0 rz 0.01 deg; joints [29.215, -45.92, 103.98, -146.801, 63.098, 164.54]
  MoveC 362 to (-267.52, 36.95, -10) mm, rotated rx -180 ry 0 rz 0.01 deg; joints [29.143, -46.018, 104.189, -146.909, 63.17, 164.645] to (-266.51, 34.19, -10) mm, rotated rx -180 ry 0 rz 0.01 deg; joints [29.07, -46.114, 104.395, -147.018, 63.241, 164.748]
  MoveC 363 to (-264.22, 31.2, -10) mm, rotated rx -180 ry 0 rz 0.01 deg; joints [29.012, -46.264, 104.715, -147.127, 63.367, 164.88] to (-260.63, 30.06, -10) mm, rotated rx 180 ry 0 rz 0.01 deg; joints [29.041, -46.426, 105.056, -147.144, 63.526, 164.975]
  MoveL 364 to (-132.88, 30.06, -10) mm, rotated rx 180 ry 0 rz 0.01 deg; joints [31.623, -51.085, 114.868, -145.686, 68.507, 166.959]
  MoveC 365 to (-129.34, 31.18, -10) mm, rotated rx 180 ry 0 rz 0.01 deg; joints [31.74, -51.185, 115.077, -145.589, 68.626, 166.979] to (-127.07, 34.12, -10) mm, rotated rx -180 ry 0 rz 0.01 deg; joints [31.894, -51.203, 115.109, -145.432, 68.676, 166.928]
  MoveC 366 to (-122.34, 45.31, -10) mm, rotated rx -180 ry 0 rz 0.01 deg; joints [32.394, -51.135, 114.943, -144.89, 68.721, 166.673] to (-116.56, 56, -10) mm, rotated rx 180 ry 0 rz 0.01 deg; joints [32.899, -51.109, 114.865, -144.355, 68.808, 166.446]
  MoveL 367 to (-104.21, 76.91, -10) mm, rotated rx 180 ry 0 rz 0.01 deg; joints [33.908, -51.08, 114.763, -143.295, 69.012, 166.013]
  MoveC 368 to (-98.15, 86.1, -10) mm, rotated rx -180 ry 0 rz 0.01 deg; joints [34.366, -51.084, 114.752, -142.819, 69.123, 165.83] to (-91.05, 94.5, -10) mm, rotated rx -180 ry 0 rz 0.01 deg; joints [34.821, -51.135, 114.844, -142.359, 69.278, 165.685]
  MoveC 369 to (-82.96, 101.98, -10) mm, rotated rx 180 ry 0 rz 0.01 deg; joints [35.27, -51.236, 115.044, -141.921, 69.478, 165.583] to (-74, 108.38, -10) mm, rotated rx -180 ry 0 rz 0.01 deg; joints [35.704, -51.387, 115.352, -141.511, 69.719, 165.526]
  MoveC 370 to (-69.46, 110.97, -10) mm, rotated rx -180 ry 0 rz 0.01 deg; joints [35.904, -51.477, 115.537, -141.329, 69.848, 165.517] to (-64.73, 113.21, -10) mm, rotated rx 180 ry 0 rz 0.01 deg; joints [36.096, -51.58, 115.752, -141.157, 69.988, 165.521]
  MoveC 371 to (-59.91, 115.24, -10) mm, rotated rx 180 ry 0 rz 0.01 deg; joints [36.284, -51.69, 115.982, -140.992, 70.132, 165.534] to (-55.06, 117.2, -10) mm, rotated rx 180 ry 0 rz 0.01 deg; joints [36.471, -51.802, 116.216, -140.828, 70.278, 165.549]
  MoveC 372 to (-52.15, 119.53, -10) mm, rotated rx -180 ry 0 rz 0.01 deg; joints [36.623, -51.843, 116.297, -140.682, 70.351, 165.522] to (-51.06, 123.09, -10) mm, rotated rx 180 ry 0 rz 0.01 deg; joints [36.771, -51.796, 116.19, -140.518, 70.346, 165.43]
  MoveL 373 to (-51.06, 274.03, -10) mm, rotated rx -180 ry 0 rz 0.01 deg; joints [41.533, -47.958, 107.835, -134.543, 68.518, 160.421]
  MoveC 374 to (-52.19, 276.75, -10) mm, rotated rx 180 ry 0 rz 0.01 deg; joints [41.584, -47.846, 107.595, -134.456, 68.446, 160.304] to (-54.91, 277.88, -10) mm, rotated rx 180 ry 0 rz 0.01 deg; joints [41.546, -47.726, 107.343, -134.457, 68.34, 160.216]
  MoveL 375 to (-84.43, 277.88, -10) mm, rotated rx -180 ry 0 rz 0.01 deg; joints [40.79, -46.755, 105.311, -134.909, 67.318, 159.697]
  MoveC 376 to (-87.69, 276.75, -10) mm, rotated rx -180 ry 0 rz 0.01 deg; joints [40.675, -46.678, 105.152, -135.001, 67.217, 159.68] to (-89.55, 273.83, -10) mm, rotated rx 180 ry 0 rz 0.01 deg; joints [40.543, -46.697, 105.196, -135.141, 67.187, 159.752]
  MoveC 377 to (-96.74, 254.45, -10) mm, rotated rx -180 ry 0 rz 0.01 deg; joints [39.791, -46.991, 105.841, -136.005, 67.163, 160.321] to (-108.39, 237.38, -10) mm, rotated rx 180 ry 0 rz 0.01 deg; joints [38.993, -47.057, 106.007, -136.844, 66.952, 160.721]
  MoveC 378 to (-123.65, 223.47, -10) mm, rotated rx -180 ry 0 rz 0.01 deg; joints [38.202, -46.904, 105.709, -137.607, 66.568, 160.94] to (-141.58, 213.24, -10) mm, rotated rx 180 ry 0 rz 0.01 deg; joints [37.465, -46.548, 104.982, -138.252, 66.035, 160.98]
  MoveC 379 to (-160.07, 207.41, -10) mm, rotated rx 180 ry 0 rz 0.01 deg; joints [36.859, -46.045, 103.941, -138.715, 65.421, 160.852] to (-179.35, 205.49, -10) mm, rotated rx -180 ry 0 rz 0.01 deg; joints [36.362, -45.399, 102.598, -139.014, 64.72, 160.567]
  MoveL 380 to (-214.91, 205.49, -10) mm, rotated rx 180 ry 0 rz 0.01 deg; joints [35.579, -44.082, 99.855, -139.373, 63.358, 159.895]
  MoveC 381 to (-231.43, 207.04, -10) mm, rotated rx -180 ry 0 rz 0.01 deg; joints [35.271, -43.412, 98.462, -139.454, 62.695, 159.515] to (-247.38, 211.61, -10) mm, rotated rx -180 ry 0 rz 0.01 deg; joints [35.072, -42.673, 96.92, -139.389, 62.011, 159.025]
  MoveC 382 to (-262.29, 218.84, -10) mm, rotated rx 180 ry 0 rz 0.01 deg; joints [34.976, -41.891, 95.288, -139.191, 61.329, 158.444] to (-275.89, 228.31, -10) mm, rotated rx -180 ry 0 rz 0.01 deg; joints [34.975, -41.087, 93.609, -138.874, 60.668, 157.788]
  MoveC 383 to (-284.59, 236.62, -10) mm, rotated rx 180 ry 0 rz 0.01 deg; joints [35.039, -40.502, 92.387, -138.568, 60.215, 157.271] to (-291.95, 246.12, -10) mm, rotated rx 180 ry 0 rz 0.01 deg; joints [35.164, -39.93, 91.192, -138.197, 59.801, 156.726]
  MoveC 384 to (-293.26, 250.53, -10) mm, rotated rx 180 ry 0 rz 0.01 deg; joints [35.264, -39.75, 90.814, -138.015, 59.695, 156.519] to (-291.88, 254.91, -10) mm, rotated rx 180 ry 0 rz 0.01 deg; joints [35.418, -39.682, 90.665, -137.823, 59.701, 156.374]
  MoveC 385 to (-290.36, 259.19, -10) mm, rotated rx -180 ry 0 rz 0.01 deg; joints [35.571, -39.621, 90.534, -137.634, 59.713, 156.236] to (-291.17, 263.66, -10) mm, rotated rx 180 ry 0 rz 0.01 deg; joints [35.682, -39.458, 90.19, -137.447, 59.627, 156.035]
  MoveC 386 to (-292.91, 268, -10) mm, rotated rx 180 ry 0 rz 0.01 deg; joints [35.769, -39.258, 89.772, -137.268, 59.504, 155.816] to (-294.16, 272.49, -10) mm, rotated rx 180 ry 0 rz 0.01 deg; joints [35.871, -39.073, 89.384, -137.08, 59.399, 155.6]
  MoveL 387 to (-296.54, 283.21, -10) mm, rotated rx -180 ry 0 rz 0.01 deg; joints [36.123, -38.654, 88.503, -136.629, 59.173, 155.096]
  MoveC 388 to (-298.36, 286.1, -10) mm, rotated rx 180 ry 0 rz 0.01 deg; joints [36.167, -38.49, 88.16, -136.51, 59.063, 154.929] to (-301.59, 287.24, -10) mm, rotated rx 180 ry 0 rz 0.01 deg; joints [36.133, -38.318, 87.806, -136.47, 58.915, 154.801]
  MoveL 389 to (-347.97, 287.23, -10) mm, rotated rx 180 ry 0 rz 0.01 deg; joints [35.21, -36.285, 83.623, -136.511, 56.934, 153.579]
  MoveC 390 to (-350.69, 286.11, -10) mm, rotated rx -180 ry 0 rz 0.01 deg; joints [35.126, -36.197, 83.444, -136.559, 56.828, 153.553] to (-351.82, 283.38, -10) mm, rotated rx -180 ry 0 rz 0.01 deg; joints [35.029, -36.231, 83.517, -136.679, 56.812, 153.643]
  MoveL 391 to (-351.82, 115.6, -10) mm, rotated rx -180 ry 0 rz 0.01 deg; joints [30.128, -40.83, 93.261, -144.034, 58.757, 160.396]
  MoveC 392 to (-350.73, 112.39, -10) mm, rotated rx 180 ry 0 rz 0.01 deg; joints [30.049, -40.953, 93.521, -144.17, 58.84, 160.536] to (-347.91, 110.52, -10) mm, rotated rx -180 ry 0 rz 0.01 deg; joints [30.041, -41.118, 93.866, -144.241, 58.983, 160.663]
  MoveC 393 to (-333.55, 105.18, -10) mm, rotated rx -180 ry 0 rz 0.01 deg; joints [30.134, -41.852, 95.394, -144.415, 59.661, 161.149] to (-320.44, 97.23, -10) mm, rotated rx 180 ry 0 rz 0.01 deg; joints [30.123, -42.582, 96.922, -144.694, 60.307, 161.69]
  MoveC 394 to (-308.96, 87.11, -10) mm, rotated rx 180 ry 0 rz 0.01 deg; joints [30.013, -43.284, 98.398, -145.064, 60.904, 162.26] to (-299.31, 75.23, -10) mm, rotated rx -180 ry 0 rz 0.01 deg; joints [29.81, -43.941, 99.785, -145.512, 61.439, 162.843]
  MoveL 395 to (-279.07, 40.39, -10) mm, rotated rx -180 ry 0 rz 0.01 deg; joints [29.044, -45.495, 103.09, -146.855, 62.659, 164.341]
  MoveC 396 to (-277.17, 36.64, -10) mm, rotated rx -180 ry 0 rz 0.01 deg; joints [28.954, -45.648, 103.415, -147.001, 62.777, 164.492] to (-275.71, 32.69, -10) mm, rotated rx -180 ry 0 rz 0.01 deg; joints [28.849, -45.787, 103.713, -147.157, 62.88, 164.642]
  MoveC 397 to (-274.43, 28.7, -10) mm, rotated rx -180 ry 0 rz 0.01 deg; joints [28.739, -45.919, 103.997, -147.318, 62.977, 164.789] to (-273.05, 24.73, -10) mm, rotated rx 180 ry 0 rz 0.01 deg; joints [28.631, -46.054, 104.286, -147.476, 63.076, 164.937]
  MoveC 398 to (-270.82, 21.81, -10) mm, rotated rx -180 ry 0 rz 0.01 deg; joints [28.574, -46.2, 104.598, -147.583, 63.199, 165.065] to (-267.31, 20.7, -10) mm, rotated rx 180 ry 0 rz 0.01 deg; joints [28.601, -46.359, 104.932, -147.601, 63.355, 165.157]
  MoveL 399 to (-126.2, 20.7, -10) mm, rotated rx 180 ry 0 rz 0.01 deg; joints [31.436, -51.503, 115.775, -145.989, 68.865, 167.326]
  MoveC 400 to (-122.67, 21.82, -10) mm, rotated rx 180 ry 0 rz 0.01 deg; joints [31.553, -51.602, 115.982, -145.89, 68.983, 167.346] to (-120.44, 24.78, -10) mm, rotated rx 180 ry 0 rz 0.01 deg; joints [31.709, -51.619, 116.012, -145.731, 69.032, 167.294]
  MoveC 401 to (-119, 28.95, -10) mm, rotated rx 180 ry 0 rz 0.01 deg; joints [31.889, -51.584, 115.929, -145.533, 69.036, 167.196] to (-117.62, 33.13, -10) mm, rotated rx -180 ry 0 rz 0.01 deg; joints [32.069, -51.546, 115.84, -145.336, 69.038, 167.097]
  MoveC 402 to (-116.05, 37.25, -10) mm, rotated rx -180 ry 0 rz 0.01 deg; joints [32.25, -51.515, 115.766, -145.138, 69.048, 167.001] to (-114.04, 41.19, -10) mm, rotated rx -180 ry 0 rz 0.01 deg; joints [32.435, -51.503, 115.731, -144.942, 69.076, 166.917]
  MoveL 403 to (-96.11, 72.22, -10) mm, rotated rx 180 ry 0 rz 0.01 deg; joints [33.935, -51.454, 115.564, -143.365, 69.362, 166.276]
  MoveC 404 to (-86.6, 85.38, -10) mm, rotated rx -180 ry 0 rz 0.01 deg; joints [34.614, -51.484, 115.603, -142.666, 69.547, 166.028] to (-74.63, 96.35, -10) mm, rotated rx 180 ry 0 rz 0.01 deg; joints [35.279, -51.637, 115.904, -142.017, 69.842, 165.882]
  MoveC 405 to (-60.78, 104.79, -10) mm, rotated rx -180 ry 0 rz 0.01 deg; joints [35.907, -51.899, 116.446, -141.435, 70.229, 165.839] to (-45.6, 110.52, -10) mm, rotated rx 180 ry 0 rz 0.01 deg; joints [36.482, -52.259, 117.198, -140.935, 70.689, 165.897]
  MoveC 406 to (-42.78, 112.42, -10) mm, rotated rx -180 ry 0 rz 0.01 deg; joints [36.618, -52.305, 117.294, -140.807, 70.764, 165.883] to (-41.69, 115.64, -10) mm, rotated rx 180 ry 0 rz 0.01 deg; joints [36.756, -52.267, 117.205, -140.656, 70.762, 165.801]
  MoveL 407 to (-41.7, 283.39, -10) mm, rotated rx -180 ry 0 rz 0.01 deg; joints [42.054, -47.997, 107.902, -134.029, 68.724, 160.246]
  MoveC 408 to (-42.83, 286.11, -10) mm, rotated rx -180 ry 0 rz 0.01 deg; joints [42.103, -47.885, 107.662, -133.944, 68.653, 160.129] to (-45.55, 287.24, -10) mm, rotated rx 180 ry 0 rz 0.01 deg; joints [42.065, -47.765, 107.41, -133.945, 68.547, 160.041]
  MoveL 409 to (-91.87, 287.24, -10) mm, rotated rx 180 ry 0 rz 0.01 deg; joints [40.876, -46.241, 104.224, -134.652, 66.946, 159.221]
  MoveC 410 to (-95.1, 286.12, -10) mm, rotated rx 180 ry 0 rz 0.01 deg; joints [40.762, -46.164, 104.065, -134.741, 66.845, 159.203] to (-96.94, 283.24, -10) mm, rotated rx -180 ry 0 rz 0.01 deg; joints [40.633, -46.184, 104.11, -134.879, 66.815, 159.276]
  MoveC 411 to (-98.4, 277.2, -10) mm, rotated rx 180 ry 0 rz 0.01 deg; joints [40.421, -46.304, 104.371, -135.135, 66.834, 159.47] to (-99.92, 271.18, -10) mm, rotated rx -180 ry 0 rz 0.01 deg; joints [40.207, -46.421, 104.624, -135.393, 66.852, 159.662]
  MoveC 412 to (-101.84, 265.26, -10) mm, rotated rx 180 ry 0 rz 0.01 deg; joints [39.985, -46.521, 104.842, -135.652, 66.854, 159.842] to (-104.44, 259.61, -10) mm, rotated rx 180 ry 0 rz 0.01 deg; joints [39.754, -46.588, 104.991, -135.91, 66.829, 159.999]
  MoveC 413 to (-109.03, 252.01, -10) mm, rotated rx 180 ry 0 rz 0.01 deg; joints [39.416, -46.64, 105.112, -136.274, 66.755, 160.19] to (-114.34, 244.91, -10) mm, rotated rx -180 ry 0 rz 0.01 deg; joints [39.074, -46.652, 105.147, -136.628, 66.65, 160.349]
  MoveC 414 to (-120.4, 238.42, -10) mm, rotated rx -180 ry 0 rz 0.01 deg; joints [38.733, -46.618, 105.087, -136.968, 66.508, 160.471] to (-127.2, 232.71, -10) mm, rotated rx 180 ry 0 rz 0.01 deg; joints [38.397, -46.536, 104.925, -137.285, 66.33, 160.551]
  MoveC 415 to (-133.76, 228.21, -10) mm, rotated rx -180 ry 0 rz 0.01 deg; joints [38.105, -46.427, 104.706, -137.551, 66.145, 160.593] to (-140.63, 224.19, -10) mm, rotated rx 180 ry 0 rz 0.01 deg; joints [37.821, -46.293, 104.432, -137.8, 65.941, 160.612]
  MoveC 416 to (-147.86, 220.83, -10) mm, rotated rx 180 ry 0 rz 0.01 deg; joints [37.55, -46.127, 104.092, -138.025, 65.715, 160.6] to (-155.42, 218.33, -10) mm, rotated rx 180 ry 0 rz 0.01 deg; joints [37.298, -45.925, 103.673, -138.218, 65.465, 160.551]
  MoveC 417 to (-170.11, 215.46, -10) mm, rotated rx 180 ry 0 rz 0.01 deg; joints [36.874, -45.474, 102.737, -138.505, 64.951, 160.384] to (-185.05, 214.64, -10) mm, rotated rx -180 ry 0 rz 0.01 deg; joints [36.512, -44.952, 101.651, -138.702, 64.397, 160.134]
  MoveL 418 to (-214.9, 214.86, -10) mm, rotated rx 180 ry 0 rz 0.01 deg; joints [35.861, -43.835, 99.327, -138.987, 63.25, 159.554]
  MoveC 419 to (-229.83, 216.26, -10) mm, rotated rx -180 ry 0 rz 0.01 deg; joints [35.582, -43.229, 98.067, -139.058, 62.651, 159.207] to (-244.22, 220.43, -10) mm, rotated rx -180 ry 0 rz 0.01 deg; joints [35.4, -42.56, 96.672, -138.999, 62.034, 158.76]
  MoveC 420 to (-257.68, 226.98, -10) mm, rotated rx 180 ry 0 rz 0.01 deg; joints [35.312, -41.853, 95.196, -138.819, 61.42, 158.232] to (-269.95, 235.55, -10) mm, rotated rx 180 ry 0 rz 0.01 deg; joints [35.308, -41.126, 93.679, -138.536, 60.825, 157.637]
  MoveC 421 to (-276.14, 241.32, -10) mm, rotated rx -180 ry 0 rz 0.01 deg; joints [35.348, -40.715, 92.82, -138.326, 60.506, 157.275] to (-281.55, 247.82, -10) mm, rotated rx -180 ry 0 rz 0.01 deg; joints [35.425, -40.311, 91.975, -138.079, 60.209, 156.896]
  MoveC 422 to (-286.27, 254.82, -10) mm, rotated rx 180 ry 0 rz 0.01 deg; joints [35.53, -39.917, 91.15, -137.803, 59.933, 156.508] to (-290.43, 262.17, -10) mm, rotated rx 180 ry 0 rz 0.01 deg; joints [35.654, -39.532, 90.345, -137.507, 59.675, 156.113]
  MoveC 423 to (-290.81, 262.91, -10) mm, rotated rx -180 ry 0 rz 0.01 deg; joints [35.668, -39.494, 90.267, -137.477, 59.651, 156.074] to (-291.17, 263.66, -10) mm, rotated rx 180 ry 0 rz 0.01 deg; joints [35.682, -39.458, 90.19, -137.447, 59.627, 156.035]
  MoveC 424 to (-291.78, 268.49, -10) mm, rotated rx 180 ry 0 rz 0.01 deg; joints [35.806, -39.291, 89.838, -137.243, 59.545, 155.823] to (-289.47, 272.77, -10) mm, rotated rx 180 ry 0 rz 0.01 deg; joints [35.974, -39.261, 89.771, -137.052, 59.59, 155.702]
  MoveC 425 to (-286.99, 276.87, -10) mm, rotated rx 180 ry 0 rz 0.01 deg; joints [36.141, -39.243, 89.728, -136.868, 59.644, 155.592] to (-286.87, 281.66, -10) mm, rotated rx 180 ry 0 rz 0.01 deg; joints [36.278, -39.106, 89.437, -136.663, 59.592, 155.397]
  MoveC 426 to (-288.02, 287.2, -10) mm, rotated rx 180 ry 0 rz 0.01 deg; joints [36.41, -38.891, 88.987, -136.431, 59.479, 155.138] to (-288.83, 292.8, -10) mm, rotated rx -180 ry 0 rz 0.01 deg; joints [36.549, -38.688, 88.56, -136.194, 59.379, 154.883]
  MoveC 427 to (-290.23, 295.51, -10) mm, rotated rx -180 ry 0 rz 0.01 deg; joints [36.596, -38.547, 88.265, -136.083, 59.289, 154.734] to (-293.08, 296.6, -10) mm, rotated rx -180 ry 0 rz 0.01 deg; joints [36.567, -38.393, 87.947, -136.045, 59.158, 154.616]
  MoveL 428 to (-357.33, 296.6, -10) mm, rotated rx 180 ry 0 rz 0.01 deg; joints [35.285, -35.564, 82.127, -136.08, 56.41, 152.894]
  MoveC 429 to (-360.05, 295.47, -10) mm, rotated rx -180 ry 0 rz 0.01 deg; joints [35.202, -35.474, 81.945, -136.125, 56.303, 152.866] to (-361.18, 292.74, -10) mm, rotated rx 180 ry 0 rz 0.01 deg; joints [35.105, -35.508, 82.019, -136.246, 56.286, 152.957]
  MoveL 430 to (-361.18, 107.29, -10) mm, rotated rx -180 ry 0 rz 0.01 deg; joints [29.705, -40.626, 92.852, -144.424, 58.44, 160.501]
  MoveC 431 to (-360.09, 104.38, -10) mm, rotated rx -180 ry 0 rz 0.01 deg; joints [29.635, -40.742, 93.098, -144.547, 58.52, 160.631] to (-357.35, 102.9, -10) mm, rotated rx 180 ry 0 rz 0.01 deg; joints [29.637, -40.895, 93.416, -144.603, 58.656, 160.742]
  MoveC 432 to (-348.81, 101.15, -10) mm, rotated rx 180 ry 0 rz 0.01 deg; joints [29.734, -41.302, 94.261, -144.651, 59.048, 160.983] to (-340.58, 98.3, -10) mm, rotated rx 180 ry 0 rz 0.01 deg; joints [29.792, -41.717, 95.127, -144.742, 59.435, 161.252]
  MoveC 433 to (-332.75, 94.48, -10) mm, rotated rx -180 ry 0 rz 0.01 deg; joints [29.813, -42.134, 95.999, -144.873, 59.814, 161.544] to (-325.4, 89.8, -10) mm, rotated rx 180 ry 0 rz 0.01 deg; joints [29.798, -42.548, 96.864, -145.039, 60.179, 161.852]
  MoveC 434 to (-320.11, 85.53, -10) mm, rotated rx -180 ry 0 rz 0.01 deg; joints [29.759, -42.863, 97.527, -145.195, 60.451, 162.103] to (-315.35, 80.67, -10) mm, rotated rx 180 ry 0 rz 0.01 deg; joints [29.691, -43.168, 98.169, -145.377, 60.705, 162.36]
  MoveC 435 to (-311.03, 75.43, -10) mm, rotated rx 180 ry 0 rz 0.01 deg; joints [29.602, -43.462, 98.788, -145.577, 60.945, 162.619] to (-307.04, 69.94, -10) mm, rotated rx 180 ry 0 rz 0.01 deg; joints [29.498, -43.745, 99.388, -145.787, 61.173, 162.879]
  MoveL 436 to (-287.16, 35.73, -10) mm, rotated rx -180 ry 0 rz 0.01 deg; joints [28.741, -45.273, 102.635, -147.116, 62.375, 164.352]
  MoveC 437 to (-284.7, 30.84, -10) mm, rotated rx -180 ry 0 rz 0.01 deg; joints [28.623, -45.472, 103.058, -147.307, 62.53, 164.549] to (-282.8, 25.72, -10) mm, rotated rx 180 ry 0 rz 0.01 deg; joints [28.486, -45.652, 103.444, -147.511, 62.664, 164.744]
  MoveC 438 to (-281.25, 20.48, -10) mm, rotated rx -180 ry 0 rz 0.01 deg; joints [28.339, -45.819, 103.804, -147.724, 62.784, 164.934] to (-279.83, 15.21, -10) mm, rotated rx 180 ry 0 rz 0.01 deg; joints [28.187, -45.981, 104.153, -147.939, 62.899, 165.122]
  MoveC 439 to (-278, 12.42, -10) mm, rotated rx 180 ry 0 rz 0.01 deg; joints [28.126, -46.109, 104.425, -148.044, 63.005, 165.239] to (-274.84, 11.34, -10) mm, rotated rx 180 ry 0 rz 0.01 deg; joints [28.146, -46.253, 104.73, -148.065, 63.147, 165.324]
  MoveL 440 to (-118.73, 11.34, -10) mm, rotated rx 180 ry 0 rz 0.01 deg; joints [31.263, -51.944, 116.733, -146.278, 69.253, 167.701]
  MoveC 441 to (-115.53, 12.42, -10) mm, rotated rx 180 ry 0 rz 0.01 deg; joints [31.372, -52.032, 116.917, -146.185, 69.359, 167.717] to (-113.64, 15.21, -10) mm, rotated rx -180 ry 0 rz 0.01 deg; joints [31.515, -52.041, 116.929, -146.038, 69.396, 167.665]
  MoveC 442 to (-108.91, 29.05, -10) mm, rotated rx -180 ry 0 rz 0.01 deg; joints [32.118, -51.924, 116.652, -145.378, 69.408, 167.342] to (-102.5, 42.2, -10) mm, rotated rx -180 ry 0 rz 0.01 deg; joints [32.732, -51.872, 116.514, -144.724, 69.487, 167.059]
  MoveL 443 to (-88, 67.54, -10) mm, rotated rx -180 ry 0 rz 0.01 deg; joints [33.961, -51.824, 116.36, -143.432, 69.711, 166.537]
  MoveC 444 to (-66.11, 91.12, -10) mm, rotated rx 180 ry 0 rz 0.01 deg; joints [35.307, -52.031, 116.753, -142.09, 70.208, 166.169] to (-36.15, 102.88, -10) mm, rotated rx -180 ry 0 rz 0.01 deg; joints [36.46, -52.732, 118.222, -141.078, 71.111, 166.271]
  MoveC 445 to (-33.42, 104.4, -10) mm, rotated rx 180 ry 0 rz 0.01 deg; joints [36.582, -52.784, 118.33, -140.965, 71.187, 166.267] to (-32.33, 107.34, -10) mm, rotated rx 180 ry 0 rz 0.01 deg; joints [36.711, -52.753, 118.256, -140.825, 71.188, 166.195]
  MoveL 446 to (-32.34, 292.75, -10) mm, rotated rx 180 ry 0 rz 0.01 deg; joints [42.574, -48.031, 107.959, -133.515, 68.928, 160.07]
  MoveC 447 to (-33.47, 295.48, -10) mm, rotated rx -180 ry 0 rz 0.01 deg; joints [42.623, -47.918, 107.717, -133.43, 68.858, 159.952] to (-36.19, 296.6, -10) mm, rotated rx -180 ry 0 rz 0.01 deg; joints [42.583, -47.799, 107.466, -133.433, 68.752, 159.864]
  MoveL 448 to (-100.46, 296.6, -10) mm, rotated rx -180 ry 0 rz 0.01 deg; joints [40.931, -45.683, 103.045, -134.406, 66.532, 158.716]
  MoveC 449 to (-103.3, 295.52, -10) mm, rotated rx 180 ry 0 rz 0.01 deg; joints [40.829, -45.618, 102.911, -134.487, 66.444, 158.704] to (-104.68, 292.81, -10) mm, rotated rx 180 ry 0 rz 0.01 deg; joints [40.717, -45.648, 102.978, -134.611, 66.427, 158.78]
  MoveC 450 to (-105.72, 285.38, -10) mm, rotated rx 180 ry 0 rz 0.01 deg; joints [40.477, -45.825, 103.357, -134.916, 66.478, 159.036] to (-107.28, 278.04, -10) mm, rotated rx -180 ry 0 rz 0.01 deg; joints [40.225, -45.979, 103.69, -135.225, 66.509, 159.278]
  MoveC 451 to (-109.55, 270.87, -10) mm, rotated rx -180 ry 0 rz 0.01 deg; joints [39.96, -46.102, 103.958, -135.537, 66.513, 159.499] to (-112.69, 264.04, -10) mm, rotated rx -180 ry 0 rz 0.01 deg; joints [39.682, -46.184, 104.141, -135.849, 66.482, 159.69]
  MoveC 452 to (-116.74, 257.32, -10) mm, rotated rx 180 ry 0 rz 0.01 deg; joints [39.385, -46.231, 104.248, -136.169, 66.416, 159.86] to (-121.42, 251.03, -10) mm, rotated rx 180 ry 0 rz 0.01 deg; joints [39.085, -46.242, 104.281, -136.48, 66.322, 160.002]
  MoveC 453 to (-126.76, 245.28, -10) mm, rotated rx 180 ry 0 rz 0.01 deg; joints [38.785, -46.213, 104.23, -136.779, 66.197, 160.111] to (-132.77, 240.23, -10) mm, rotated rx 180 ry 0 rz 0.01 deg; joints [38.49, -46.14, 104.086, -137.058, 66.039, 160.183]
  MoveC 454 to (-138.61, 236.22, -10) mm, rotated rx 180 ry 0 rz 0.01 deg; joints [38.232, -46.044, 103.892, -137.292, 65.873, 160.221] to (-144.7, 232.62, -10) mm, rotated rx 180 ry 0 rz 0.01 deg; joints [37.98, -45.926, 103.651, -137.512, 65.692, 160.238]
  MoveC 455 to (-151.12, 229.61, -10) mm, rotated rx 180 ry 0 rz 0.01 deg; joints [37.739, -45.779, 103.35, -137.712, 65.491, 160.228] to (-157.85, 227.37, -10) mm, rotated rx 180 ry 0 rz 0.01 deg; joints [37.515, -45.599, 102.979, -137.882, 65.269, 160.185]
